(* Logix 5000 project; controller R5_CSS vendor 1 type 14 code 74 rev 19.11; software revision 19.01 *)
// Condensing System

TASK MainTask (continuous, watchdog 500 ms) : MainProgram
TASK MSG (periodic, rate 500 ms, priority 10, watchdog 1000 ms) : POD1_MSG
TASK PIDE (periodic, rate 10 ms, priority 10, watchdog 500 ms) : PIDE   // Advanced PID operations for most important control loops

MODULES
   Local : vendor 1 type 14 code 74 (Compact 0, 1768Ctrl5Slot 0, rev 19.11)
      SLOT_2 : vendor 1 type 7 code 69 (Compact 2, rev 3.1, Input RPI 20 ms)
           Local:2:I.DATA.10   // P205 OVERHEAD CONDENSER PUMP RUN STATUS
      SLOT_3 : vendor 1 type 7 code 69 (Compact 3, rev 3.1, Input RPI 20 ms)
           Local:3:I.DATA.6   // PRIMARY COALESCER SEPARATOR TEMPERATURE CONTROL RUN STATUS
      MVI69 : 1769-MODULE (Compact 1, rev 1.1, Output RPI 2 ms)
      SLOT_11 : 1769-IF8 (Compact 11, rev 1.1, Output RPI 80 ms)
           Local:11:I.CH0DATA   // QUENCH BASIN FLOW TRANSMITTER
           Local:11:I.CH1DATA   // QUENCH FEED FLOW TRANSMITTER
           Local:11:I.CH2DATA   // QUENCH CONDITIONING QUENCH WATER PHASE FLOW TRANSMITTER
           Local:11:I.CH3DATA   // QUENCH TOWER UPPER SPRAY FIT
           Local:11:I.CH4DATA   // QUENCH TOWER LOWER SPRAY FLOW TRANSMITTER
           Local:11:I.CH5DATA   // QUENCH TOWER BASIN LEVEL TRANSMITTER
           Local:11:I.CH6DATA   // QUENCH COALESCING SEPARATOR SECONDARY CHAMBER LEVEL TRANSMITTER
      SLOT_10 : 1769-IF8 (Compact 10, rev 1.1, Output RPI 80 ms)
           Local:10:I.CH3DATA   // QUENCH WATER CONDUCTIVITY TRANSMITTER
           Local:10:I.CH0DATA   // QUENCH BASIN TRANSFER BASIN B TEMPERATURE TRANSMITTER
           Local:10:I.CH1DATA   // COALESCER OIL CHAMBER SHELL TEMPERATURE TRANSMITTER
      SLOT_7 : 1769-IF8 (Compact 7, rev 1.1, Output RPI 80 ms)
           Local:7:I.CH0DATA   // QUENCH TOWER EXIT GAS TEMPERATURE TRANSMITTER
           Local:7:I.CH1DATA   // GTL FROM PRUA TEMPERATURE TRANSMITTER
           Local:7:I.CH2DATA   // GTL FROM PRUB TEMPERATURE TRANSMITTER
           Local:7:I.CH3DATA   // GTL FROM PRUC TEMPERATURE TRANSMITTER
           Local:7:I.CH4DATA   // GTL FROM PRUD TEMPERATURE TRANSMITTER
           Local:7:I.CH5DATA   // HEAT JACKET VENT FROM PRUA TEMPERATURE TRANSMITTER
           Local:7:I.CH6DATA   // HEAT JACKET VENT FROM PRUB TEMPERATURE TRANSMITTER
           Local:7:I.CH7DATA   // HEAT JACKET VENT FROM PRUC TEMPERATURE TRANSMITTER
      SLOT_8 : 1769-IF8 (Compact 8, rev 1.1, Output RPI 80 ms)
           Local:8:I.CH4DATA   // PRIMARY COALESCER SEPARATOR TEMPERATURE TRANSMITTER
           Local:8:I.CH0DATA   // HEAT JACKET VENT FROM PRUD TEMPERATURE TRANSMITTER
           Local:8:I.CH1DATA   // PROCESS WATER POST HX TEMPERATURE TRANSMITTER
           Local:8:I.CH2DATA   // HX COOLING WATER SUPPLY TEMPERATURE TRANSMITTER
           Local:8:I.CH3DATA   // HX COOLING WATER RETURN TEMPERATURE TRANSMITTER
           Local:8:I.CH5DATA   // PRIMARY COALESCER SHELL TEMPERATURE TRANSMITTER
           Local:8:I.CH6DATA   // QUENCH BASIN LIQUID TEMPERATURE TRANSMITTER
           Local:8:I.CH7DATA   // QUENCH BASIN SHELL TEMPERATURE TRANSMITTER
      SLOT_13 : vendor 1 type 10 code 40 (Compact 13, rev 2.1, Output RPI 80 ms)
      SLOT_12 : vendor 1 type 10 code 40 (Compact 12, rev 2.1, Output RPI 80 ms)
      SLOT_4 : 1769-IF8 (Compact 4, rev 1.1, Output RPI 80 ms)
           Local:4:I.CH0DATA   // COALESCER PROCESS IMPURITY FLOW RAW IMPUT
           Local:4:I.CH1DATA   // COALESCER MAKE UP WATER RAW IMPUT
           Local:4:I.CH2DATA   // LOWER QUENCH TOWER PRESSURE TRANSMITTER RAW INPUT
           Local:4:I.CH3DATA   // UPPER QUENCH TOWER PRESSURE TRANSMITTER RAW INPUT
           Local:4:I.CH4DATA   // QUENCH BASIN TRANSFER PUMP SUCTION PRESSURE INDICATOR RAW INPUT
           Local:4:I.CH5DATA   // QUENCH BASIN TRANSFER PUMP DISCHARGE PRESSURE RAW INPUT
           Local:4:I.CH6DATA   // PRE HX LOW PRESSURE TRANSMITTER RAW INPUT
           Local:4:I.CH7DATA   // POST HX LOW PRESSURE TRANSMITTER RAW INPUT
      SLOT_9 : 1769-IF8 (Compact 9, rev 1.1, Output RPI 80 ms)
           Local:9:I.CH0DATA   // OVERHEAD CONDENSER CHILLED WATER TEMPERATURE TRANSMITTER
           Local:9:I.CH1DATA   // OVERHEAD CONDENSER BASIN TEMPERATURE TRANSMITTER
           Local:9:I.CH2DATA   // OVERHEAD CONDENSER CHILLED WATER SUPPLY TEMPERATURE
           Local:9:I.CH3DATA   // OVERHEAD CONDENSED CHILLED WATER RETURN TEMPERATURE TRANSMITTER
           Local:9:I.CH4DATA   // COALESCER OIL CHAMBER SHELL TEMPERATURE TRANSMITTER
           Local:9:I.CH5DATA   // COALESCER OIL CHAMBER TRANSFER PUMP A TEMPERATURE TRANSMITTER
           Local:9:I.CH6DATA   // COALESCER OIL CHAMBER TRANSFER PUMP B TEMPERATURE TRANSMITTER
           Local:9:I.CH7DATA   // QUENCH BASIN TRANSFER BASIN A TEMPERATURE TRANSMITTER
      SLOT_5 : 1769-IF8 (Compact 5, rev 1.1, Output RPI 80 ms)
           Local:5:I.CH4DATA   // VACUUM SYSTEM PRESSURE TRANSMITTER RAW INPUT
           Local:5:I.CH5DATA   // HX COOLING WATER FLOW TRANMITTER
           Local:5:I.CH6DATA   // OVERHEAD CONDENSER CHILLED WATER FLOW TRANSMITTER RAW INPUT
           Local:5:I.CH7DATA   // VENT HEADER PRESSURE TRANSMITTER RAW INPUT
      SLOT_14 : vendor 1 type 7 code 73 (Compact 14, rev 3.1, Output RPI 20 ms)
           Local:14:O.DATA.4   // HS302B P302B Oil Transfer Pump Start Relay
           Local:14:O.DATA.5   // HS205 P205 Overhead Condenser Basin Transfer Start
           Local:14:O.DATA.25   // MP-113 Start
           Local:14:O.DATA.26   // Alarm Horn (Future)
           Local:14:O.DATA.12   // FCV141 PLANT RAW WATER INLET TO QUENCH TOWER ENERGIZE TO OPEN
           Local:14:O.DATA.0   // Loss of Panel Purge Indicator Light
           Local:14:O.DATA.1   // Spare
           Local:14:O.DATA.2   // Spare
           Local:14:O.DATA.14   // HS104B Valve P101B Quench Transfer FAIL OPEN ENERGISE TO CLOSE
           Local:14:O.DATA.16   // HS313 Primary Settler Heat Controller
           Local:14:O.DATA.3   // HS302A P302A Oil Transfer Pump Start Relay
           Local:14:O.DATA.7   // HS_MP112 Quench Transfer Metal Treat Meter Pump #2 Start
           Local:14:O.DATA.6   // HS_MP113 Quench Transfer Metal Treat Meter Pump #1 Start
           Local:14:O.DATA.17   // JC306 or HS306A OIL CHAMBER SETTLER HEAT OUTPUT START
           Local:14:O.DATA.9   // HS_MP411 Quench Condition Metal Treat Meter Pump #2 Start (future)
           Local:14:O.DATA.8   // HS_MP410 Quench Condition Metal Treat Meter Pump #1 Start (future)
           Local:14:O.DATA.10   // HS315A VALVE P303A DISCHARGE FAIL OPEN ENERGIZE TO CLOSE
           Local:14:O.DATA.11   // HS315B VALVE P303B DISCHARGE FAIL OPEN ENERGIZE TO CLOSE
           Local:14:O.DATA.13   // HS104A Valve P101A Quench Transfer FAIL OPEN ENERGISE TO CLOSE
           Local:14:O.DATA.15   // Spare
           Local:14:O.DATA.18   // HS114B Quench Tower Heat Controller Hand Switch
           Local:14:O.DATA.20   // HS433B Valve HX B COOLING WATER ENERGIZE TO CLOSE
           Local:14:O.DATA.22   // HS431B Inlet Valve HX B PROCESS ENERGIZE TO CLOSE
           Local:14:O.DATA.21   // HS431A Inlet Valve HX A PROCESS ENERGIZE TO CLOSE
           Local:14:O.DATA.19   // HS433A Valve HX A COOLING WATER ENERGIZE TO CLOSE
           Local:14:O.DATA.23   // FCV410 Quench Basin Level Transmitter Hot Water Flush
           Local:14:O.DATA.24   // MV361 Sec/Ter Coalsce Chamber CrossOver Valve H3 Occupancy
           Local:14:O.DATA.27   // MV115B Basin Water Heater Valve
      SLOT_6 : 1769-IF8 (Compact 6, rev 1.1, Output RPI 80 ms)
           Local:6:I.CH0DATA   // OVERHEAD CONDENSER BASIN LEVEL TRANSMITTER RAW INPUT
           Local:6:I.CH1DATA   // COALESCER OIL CHAMBER LEVEL TRANSMITTER RAW INPUT
           Local:6:I.CH3DATA   // OVERHEAD CONDENSER CHILLED WATER TEMPERATURE TRANSMITTER RAW INPUT
      CSS_ENET : 1768-ENBT (1768 1, Ethernet 192.168.20.70, rev 4.1)
         P303B : ETHERNET-MODULE (Ethernet 192.168.20.75, rev 1.1, Output RPI 10 ms)
              P303B:I.DATA[2]   // Status Bits (Continued)
              P303B:I.DATA[2].9   // Local/Remote Keypad Status 0=Local 1-=Remote
              P303B:I.DATA[1]   // Current RPM
              P303B:I.DATA[0].0   // Faulted
              P303B:I.DATA[0].1   // Warning
              P303B:I.DATA[0].2   // Running in Forward
              P303B:I.DATA[0].3   // Running in Reverse
              P303B:I.DATA[0].4   // Ready
              P303B:I.DATA[0].5   // Ctrl from Net
              P303B:I.DATA[0].6   // Ref from Net
              P303B:I.DATA[0].7   // At Reference
              P303B:I.DATA[0]   // Status Bits
              P303B:I.DATA   // Instance 171
              P303B:I.DATA[4]   // Current Amps
              P303B:O.DATA   // Instance 21
              P303B:O.DATA[0]   // Command Bits
              P303B:O.DATA[0].0   // Run Forward Command
              P303B:O.DATA[0].1   // Run Reverse Command
              P303B:O.DATA[0].2   // Fault Reset
              P303B:O.DATA[1]   // RPM Speed Refernce
         P303A : ETHERNET-MODULE (Ethernet 192.168.20.74, rev 1.1, Output RPI 10 ms)
              P303A:I.DATA[0]   // Status Bits
              P303A:I.DATA   // Instance 171
              P303A:I.DATA[1]   // Current RPM
              P303A:I.DATA[2]   // Status Bits (Continued)
              P303A:I.DATA[4]   // Current Amps
              P303A:I.DATA[0].0   // Faulted
              P303A:I.DATA[0].1   // Warning
              P303A:I.DATA[0].2   // Running in Forward
              P303A:I.DATA[0].3   // Running in Reverse
              P303A:I.DATA[0].4   // Ready
              P303A:I.DATA[0].5   // Ctrl from Net
              P303A:I.DATA[0].6   // Ref from Net
              P303A:I.DATA[0].7   // At Reference
              P303A:I.DATA[2].9   // Local/Remote Keypad Status 0=Local 1-=Remote
              P303A:O.DATA   // Instance 21
              P303A:O.DATA[0]   // Command Bits
              P303A:O.DATA[0].1   // Run Reverse Command
              P303A:O.DATA[0].2   // Fault Reset
              P303A:O.DATA[1]   // RPM Speed Reference
              P303A:O.DATA[0].0   // Run Forward Command
         P101A : ETHERNET-MODULE (Ethernet 192.168.20.72, rev 1.1, Output RPI 10 ms)
              P101A:I.DATA[2]   // Status Bits (Continued)
              P101A:I.DATA[4]   // Current Amps
              P101A:I.DATA[0].5   // Ctrl from Net
              P101A:I.DATA[0].3   // Running In Reverse
              P101A:I.DATA[0].2   // Running In Forward
              P101A:I.DATA[0]   // Status Bits
              P101A:I.DATA   // Instance 171
              P101A:I.DATA[0].0   // Faulted
              P101A:I.DATA[0].1   // Warning
              P101A:I.DATA[0].4   // Ready
              P101A:I.DATA[0].6   // Ref from Net
              P101A:I.DATA[0].7   // At Refernce
              P101A:I.DATA[1]   // Current RPM
              P101A:I.DATA[2].9   // Local/Remote Keypad Status 0=Local 1=Remote
              P101A:O.DATA[0].8   // na
              P101A:O.DATA[1]   // RPM Speed Reference
              P101A:O.DATA[0].0   // Run Forward Command
              P101A:O.DATA[0].1   // Run Reverse Command
              P101A:O.DATA[0].2   // Fault Reset
              P101A:O.DATA[0].5   // NetCtrl
              P101A:O.DATA[0]   // Command Bits
              P101A:O.DATA[0].6   // NetRef
              P101A:O.DATA[0].10   // na
              P101A:O.DATA[0].9   // na
              P101A:O.DATA[0].11   // na
              P101A:O.DATA[0].12   // na
              P101A:O.DATA[0].13   // na
              P101A:O.DATA[0].14   // na
              P101A:O.DATA[0].15   // na
              P101A:O.DATA[0].7   // na
              P101A:O.DATA[0].4   // na
              P101A:O.DATA[0].3   // na
              P101A:O.DATA   // Instance 21
         P101B : ETHERNET-MODULE (Ethernet 192.168.20.73, rev 1.1, Output RPI 10 ms)
              P101B:I.DATA   // Instance 171
              P101B:I.DATA[0]   // Status Bits
              P101B:I.DATA[0].0   // Faulted
              P101B:I.DATA[0].1   // Warning
              P101B:I.DATA[0].2   // Running in Forward
              P101B:I.DATA[0].3   // Running in Reverse
              P101B:I.DATA[0].4   // Ready
              P101B:I.DATA[0].5   // Ctrl from Net
              P101B:I.DATA[0].6   // Ref from Net
              P101B:I.DATA[0].7   // At Reference
              P101B:I.DATA[1]   // Current RPM
              P101B:I.DATA[2]   // Status Bits (Continued)
              P101B:I.DATA[4]   // Current Amps
              P101B:I.DATA[2].9   // Local/Remote Keypad Status 0=Local 1=Remote
              P101B:O.DATA[1]   // RPM Speed Reference
              P101B:O.DATA[0]   // Command Bits
              P101B:O.DATA[0].0   // Run Forward Command
              P101B:O.DATA[0].1   // Run Reverse Command
              P101B:O.DATA[0].2   // Fault Reset
              P101B:O.DATA   // Instance 21
END_MODULES

TYPE AnalogControl :
STRUCT
   AUTO : BOOL;
   MANUAL : BOOL;
   MAN_SP : REAL;
   AUTO_SP : REAL;
   CO : REAL;
   FB : REAL;
   PID_CO : REAL;
   PV_SETPOINT : REAL;
   PV : REAL;
   HC_FAULT : BOOL;
   RUN_STATUS : BOOL;   // Boolean feedback of the running status of the associated output
   START : BOOL;   // Master logical bit used to enable an associated output
   XA_Low : BOOL;   // Signal failure (Low counts)
   XA_High : BOOL;   // Signal failure (High counts)
   RawCounts : DINT;   // Raw integer from input card
   FailMode : DINT;   // 0=raw, 1=hold last, 2=safe state
   SafeState : REAL;   // Used to hold an analog value in the event of a failed instrument
   AI_Anal : AI_Analysis;   // Used to manage an analog input to determine scaled value and loss of signal alarms
   InputMin : DINT;   // Input card lower counts i.e. 4mA - 4000 counts
   InputMax : DINT;   // Input card upper counts i.e. 20mA - 20000 counts
   ScaledMin : REAL;   // Analog low Engineering unit i.e. 4mA - 0 psi
   ScaledMax : REAL;   // Analog High Engineering unit i.e. 20mA - 100 psi
   OutputMin : DINT;   // Output card lower counts i.e. 4mA - 4000 counts
   OutputMax : DINT;   // Output card upper counts i.e. 4mA - 4000 counts
   AlarmsSetDetaults : BOOL;   // reloads the default alarm limits and setup
   Simulate : BOOL;   // 0=raw counts from Input card, 1=simulation raw counts
   RawCountsSim : DINT;   // raw count simulation from HMI/Programmer
   DifferenceExists : BOOL;
   LoadDefaults : BOOL;
   StoreDefaults : BOOL;
END_STRUCT
END_TYPE

TYPE ANALYTICAL :
STRUCT
   AUTO : BOOL;
   MANUAL : BOOL;
   MAN_SP : REAL;
   AUTO_SP : REAL;
   CO : REAL;
   FB : REAL;
   PID_CO : REAL;
   PV_SETPOINT : REAL;
   AT : REAL;
   AALL_SP : REAL;
   AAL_SP : REAL;
   AAH_SP : REAL;
   AAHH_SP : REAL;
   ALL_DEV : REAL;
   AL_DEV : REAL;
   AH_DEV : REAL;
   AHH_DEV : REAL;
   AALL : BOOL;
   AAL : BOOL;
   AAH : BOOL;
   AAHH : BOOL;
   ALL_TMR : TIMER;
   AL_TMR : TIMER;
   AH_TMR : TIMER;
   AHH_TMR : TIMER;
   XA : BOOL;   // LOSS OF SIGNAL
   Forced : BOOL;   // Override actual signal with forced value
   ForcedValue : REAL;   // used with the Forced bit
   XA_Low : BOOL;   // Signal failure (Low counts)
   XA_High : BOOL;   // Signal failure (High counts)
   RawCounts : DINT;   // Raw integer from input card
   FailMode : DINT;   // 0=raw, 1=hold last, 2=safe state
   SafeState : REAL;   // Used to hold an analog value in the event of a failed instrument
   AI_Anal : AI_Analysis;   // Used to manage an analog input to determine scaled value and loss of signal alarms
   InputMin : DINT;   // Input card lower counts i.e. 4mA - 4000 counts
   InputMax : DINT;   // Input card upper counts i.e. 20mA - 20000 counts
   ScaledMin : REAL;   // Analog low Engineering unit i.e. 4mA - 0 psi
   ScaledMax : REAL;   // Analog High Engineering unit i.e. 20mA - 100 psi
   OutputMin : DINT;   // Output card lower counts i.e. 4mA - 4000 counts
   OutputMax : DINT;   // Output card upper counts i.e. 4mA - 4000 counts
   AlarmsSetDetaults : BOOL;   // reloads the default alarm limits and setup
   Simulate : BOOL;   // 0=raw counts from Input card, 1=simulation raw counts
   RawCountsSim : DINT;   // raw count simulation from HMI/Programmer
   DifferenceExists : BOOL;   // 0 - current settings are equal to default 1 = current settings differ from default
   LoadDefaults : BOOL;   // set to 1 to load from default settings
   StoreDefaults : BOOL;   // set to 1 to save current settings into default placeholder
   PV : REAL;   // Real signal from instrument in engineering units
END_STRUCT
END_TYPE

TYPE FAULTRECORD :
STRUCT
   TIMELOW : DINT;
   TIMEHIGH : DINT;
   TYPE : INT;
   CODE : INT;
   INFO : DINT[8];
END_STRUCT
END_TYPE

TYPE FLOW_CONTROL :
STRUCT
   AUTO : BOOL;
   MANUAL : BOOL;
   MAN_SP : REAL;
   AUTO_SP : REAL;
   CO : REAL;
   FB : REAL;
   PID_CO : REAL;
   PV_SETPOINT : REAL;
   FT : REAL;
   FALL_SP : REAL;
   FAL_SP : REAL;
   FAH_SP : REAL;
   FAHH_SP : REAL;
   FALL_DEV : REAL;
   FAL_DEV : REAL;
   FAH_DEV : REAL;
   FAHH_DEV : REAL;
   FALL : BOOL;
   FAL : BOOL;
   FAH : BOOL;
   FAHH : BOOL;
   FALL_TMR : TIMER;
   FAL_TMR : TIMER;
   FAH_TMR : TIMER;
   FAHH_TMR : TIMER;
   XA : BOOL;   // OUT OF RANGE (LOW)
   Forced : BOOL;   // Override actual signal with forced value
   ForcedValue : REAL;   // used with the Forced bit
   XA_Low : BOOL;   // Signal failure (Low counts)
   XA_High : BOOL;   // Signal failure (High counts)
   RawCounts : DINT;   // Raw integer from input card
   FailMode : DINT;   // 0=raw, 1=hold last, 2=safe state
   SafeState : REAL;   // Used to hold an analog value in the event of a failed instrument
   AI_Anal : AI_Analysis;   // Used to manage an analog input to determine scaled value and loss of signal alarms
   InputMin : DINT;   // Input card lower counts i.e. 4mA - 4000 counts
   InputMax : DINT;   // Input card upper counts i.e. 20mA - 20000 counts
   ScaledMin : REAL;   // Analog low Engineering unit i.e. 4mA - 0 psi
   ScaledMax : REAL;   // Analog High Engineering unit i.e. 20mA - 100 psi
   OutputMin : DINT;   // Output card lower counts i.e. 4mA - 4000 counts
   OutputMax : DINT;   // Output card upper counts i.e. 4mA - 4000 counts
   AlarmsSetDetaults : BOOL;   // reloads the default alarm limits and setup
   Simulate : BOOL;   // 0=raw counts from Input card, 1=simulation raw counts
   RawCountsSim : DINT;   // raw count simulation from HMI/Programmer
   DifferenceExists : BOOL;   // 0 - current settings are equal to default 1 = current settings differ from default
   LoadDefaults : BOOL;   // set to 1 to load from default settings
   StoreDefaults : BOOL;   // set to 1 to save current settings into default placeholder
   PV : REAL;   // Real signal from instrument in engineering units
END_STRUCT
END_TYPE

TYPE HARTAutoPoll :
STRUCT
   Auto_Poll_CMD_Status : SINT;
   Last_Status_Byte : SINT;
   Last_Second_Status_Byte : SINT;
   Manufacture_ID_Code : SINT;
   Device_Type_Code : SINT;
   Min_Preambles : SINT;
   Universal_CMD_Major : SINT;
   Device_Rev_Level : SINT;
   Software_Rev_Level : SINT;
   Hardware_Rev_Level : SINT;
   Device_Flags : SINT;
   Device_ID : SINT[3];
   Min_Preambles_Resp : SINT;
   Max_Number_Devices : SINT;
   Config_Change_Count : INT;
   Ext_Dev_Status : SINT;
   Primary_Var_Units : SINT;
   Secondary_Var_Units : SINT;
   Tertiary_Var_Units : SINT;
   Quaternary_Var_Units : SINT;
   Tag_Name : SINT[8];
   Descriptor : SINT[16];
   Tag_Descriptor_Data : SINT[3];
   Transd_Serial_Num : SINT[3];
   Transd_limits : SINT;
   PV_Alarms : SINT;
   PV_Transfer : SINT;
   PV_URLLRV_Units : SINT;
   Write_Protection_Code : SINT;
   Private_Label_Code : SINT;
   PV_Analog_Ch_Flag : SINT;
   PV_value : REAL;
   SV_value : REAL;
   TV_value : REAL;
   QV_value : REAL;
   U_trans_limit : REAL;
   L_trans_limit : REAL;
   Min_span : REAL;
   PV_URV : REAL;
   PV_LRV : REAL;
   PV_damp : REAL;
END_STRUCT
END_TYPE

TYPE HARTBackplane :
STRUCT
   LastRead : INT;
   LastWrite : INT;
   BlockIndex : INT;
END_STRUCT
END_TYPE

TYPE HARTCHStat :
STRUCT
   State : INT;
   Comm_State : INT;
   Dev_stat : INT;
   Dev_in_poll : INT;
   Dev_long : INT;
   Cur_cmd : INT;
   Cmd_req : INT;
   Cmd_resp : INT;
   Cfg_Err : INT;
   CurErr : INT;
   LastErr : INT;
END_STRUCT
END_TYPE

TYPE HARTData :
STRUCT
   HART_IN_Float_vals : REAL[100];
   HART_IN_Int_vals : INT[500];
   HART_OUT_Float_vals : REAL[100];
   HART_OUT_Int_vals : INT[500];
END_STRUCT
END_TYPE

TYPE HARTModuleDef :
STRUCT
   GenStat : HARTStat;
   BP : HARTBackplane;
   Auto_Poll : HARTAutoPoll[10];
   ByteData : SINT[1000];
   BlockTransferSize : INT;
END_STRUCT
END_TYPE

TYPE HARTStat :
STRUCT
   Scan_Cnt : INT;
   Product_Name : SINT[4];
   Rev_Level : SINT[4];
   Op_Sys : SINT[4];
   Run_Number : SINT[4];
   Blk_Rd_Count : INT;
   Blk_Wr_Count : INT;
   Blk_Parse_Cnt : INT;
   Blk_Resv : INT;
   Blk_Cmd : INT;
   Blk_Err : INT;
   ChStat : HARTCHStat[2];
END_STRUCT
END_TYPE

TYPE IP :
STRUCT
   IP1 : SINT;
   IP2 : SINT;
   IP3 : SINT;
   IP4 : SINT;
   SN1 : SINT;
   SN2 : SINT;
   SN3 : SINT;
   SN4 : SINT;
   GW1 : SINT;
   GW2 : SINT;
   GW3 : SINT;
   GW4 : SINT;
   PNS1 : SINT;
   PNS2 : SINT;
   PNS3 : SINT;
   PNS4 : SINT;
   SNS1 : SINT;
   SNS2 : SINT;
   SNS3 : SINT;
   SNS4 : SINT;
   EMPTY : INT;
   DN : SINT[48];
END_STRUCT
END_TYPE

TYPE LEVEL_CONTROL :
STRUCT
   AUTO : BOOL;
   MANUAL : BOOL;
   MAN_SP : REAL;
   AUTO_SP : REAL;   // PUMP START SET POINT
   CO : REAL;
   FB : REAL;
   PID_CO : REAL;
   PV_SETPOINT : REAL;
   LT : REAL;
   LALL_SP : REAL;
   LAL_SP : REAL;
   LAH_SP : REAL;
   LAHH_SP : REAL;
   LDAH_SP : REAL;   // LDAH SETPOING
   LALL_DEV : REAL;
   LAL_DEV : REAL;
   LAH_DEV : REAL;
   LAHH_DEV : REAL;
   LDAH_DEV : REAL;   // LDAH DEVIATION
   LDAH_DIFF : REAL;   // LDAH DIFFERENCE
   LALL : BOOL;
   LAL : BOOL;
   LAH : BOOL;
   LAHH : BOOL;
   LDAH : BOOL;   // HIGH DIFFERENTIAL
   LALL_TMR : TIMER;
   LAL_TMR : TIMER;
   LAH_TMR : TIMER;
   LAHH_TMR : TIMER;
   LDAH_TMR : TIMER;   // HIGH DIFFERENTIAL TIMVER
   XA : BOOL;   // OUT OF RANGE SIGNAL
   Forced : BOOL;   // Override actual signal with forced value
   ForcedValue : REAL;   // used with the Forced bit
   XA_Low : BOOL;   // Signal failure (Low counts)
   XA_High : BOOL;   // Signal failure (High counts)
   RawCounts : DINT;   // Raw integer from input card
   FailMode : DINT;   // 0=raw, 1=hold last, 2=safe state
   SafeState : REAL;   // Used to hold an analog value in the event of a failed instrument
   AI_Anal : AI_Analysis;   // Used to manage an analog input to determine scaled value and loss of signal alarms
   InputMin : DINT;   // Input card lower counts i.e. 4mA - 4000 counts
   InputMax : DINT;   // Input card upper counts i.e. 20mA - 20000 counts
   ScaledMin : REAL;   // Analog low Engineering unit i.e. 4mA - 0 psi
   ScaledMax : REAL;   // Analog High Engineering unit i.e. 20mA - 100 psi
   OutputMin : DINT;   // Output card lower counts i.e. 4mA - 4000 counts
   OutputMax : DINT;   // Output card upper counts i.e. 4mA - 4000 counts
   AlarmsSetDetaults : BOOL;   // reloads the default alarm limits and setup
   Simulate : BOOL;   // 0=raw counts from Input card, 1=simulation raw counts
   RawCountsSim : DINT;   // raw count simulation from HMI/Programmer
   DifferenceExists : BOOL;   // 0 - current settings are equal to default 1 = current settings differ from default
   LoadDefaults : BOOL;   // set to 1 to load from default settings
   StoreDefaults : BOOL;   // set to 1 to save current settings into default placeholder
   PV : REAL;   // Real signal from instrument in engineering units
END_STRUCT
END_TYPE

TYPE MAJOR_FAULT :
STRUCT
   TYPE : INT;
   CODE : INT;
   INFO : DINT[8];   // [0] = Task [1] = Program [2] = Routine [3] = Address [4]-[7] not used
END_STRUCT
END_TYPE

TYPE MSG_CommsPath :
STRUCT
   Prefix : STRING;   // This is the standard hex prefix to be used to build the path
   NodeNum : DINT;   // This is the configurable node number
   NodeStr : STRING;   // this is the node number represented as a string
   Path : STRING;   // this is the complete path
END_STRUCT
END_TYPE

TYPE PRESSURE_CONTROL :
STRUCT
   AUTO : BOOL;
   MANUAL : BOOL;
   MAN_SP : REAL;
   AUTO_SP : REAL;
   CO : REAL;
   FB : REAL;
   PID_CO : REAL;
   PV_SETPOINT : REAL;
   PT : REAL;
   PDAHH_DIFF : REAL;   // PDAHH DIFFERENCE
   PDAH_DIFF : REAL;   // PDAH DIFFERENCE
   PALL_SP : REAL;
   PAL_SP : REAL;
   PAH_SP : REAL;
   PAHH_SP : REAL;
   PDAH_SP : REAL;   // HIGH DIFFERENTIAL SETPOINT
   PDAHH_SP : REAL;   // PDAHH DIFF SP
   PALL_DEV : REAL;
   PAL_DEV : REAL;
   PAH_DEV : REAL;
   PAHH_DEV : REAL;
   PDAH_DEV : REAL;   // HIGH DIFFERENTIAL ALARM CLEAR
   PDAHH_DEV : REAL;   // HI HI DIFFERENTIAL ALARM CLEAR
   PALL : BOOL;
   PAL : BOOL;
   PAH : BOOL;
   PAHH : BOOL;
   PDAH : BOOL;   // HIGH DIFFERENTIAL ALARM
   PDAHH : BOOL;   // DIFFERENTIAL ALARM HI HI
   PALL_TMR : TIMER;
   PAL_TMR : TIMER;
   PAH_TMR : TIMER;
   PDAH_TMR : TIMER;   // HIGH DIFFERENTIAL DEBOUNCE TIMER
   PAHH_TMR : TIMER;
   PDAHH_TMR : TIMER;   // HI HI DIFFERENTIAL DEBOUNCE TIMER
   XA : BOOL;   // LOSS OF SIGNAL
   XA_Low : BOOL;   // Signal failure (Low counts)
   XA_High : BOOL;   // Signal failure (High counts)
   RawCounts : DINT;   // Raw integer from input card
   FailMode : DINT;   // 0=raw, 1=hold last, 2=safe state
   SafeState : REAL;   // Used to hold an analog value in the event of a failed instrument
   AI_Anal : AI_Analysis;   // Used to manage an analog input to determine scaled value and loss of signal alarms
   InputMin : DINT;   // Input card lower counts i.e. 4mA - 4000 counts
   InputMax : DINT;   // Input card upper counts i.e. 20mA - 20000 counts
   ScaledMin : REAL;   // Analog low Engineering unit i.e. 4mA - 0 psi
   ScaledMax : REAL;   // Analog High Engineering unit i.e. 20mA - 100 psi
   OutputMin : DINT;   // Output card lower counts i.e. 4mA - 4000 counts
   OutputMax : DINT;   // Output card upper counts i.e. 4mA - 4000 counts
   AlarmsSetDetaults : BOOL;   // reloads the default alarm limits and setup
   Simulate : BOOL;   // 0=raw counts from Input card, 1=simulation raw counts
   RawCountsSim : DINT;   // raw count simulation from HMI/Programmer
   DifferenceExists : BOOL;   // 0 - current settings are equal to default 1 = current settings differ from default
   LoadDefaults : BOOL;   // set to 1 to load from default settings
   StoreDefaults : BOOL;   // set to 1 to save current settings into default placeholder
   PV : REAL;   // Real signal from instrument in engineering units
END_STRUCT
END_TYPE

TYPE PUMP_CONTROL :
STRUCT
   QAS_IAS : BOOL;
   QI_AUTO : BOOL;
   QI_MANUAL : BOOL;
   QI_LEAD : BOOL;   // LEAD STATUS
   QI_TRANSFER_LEAD : BOOL;   // HMI REQUEST LEAD
   QI_RUN_STATUS : BOOL;
   START : BOOL;
   LAL_ENABLE : BOOL;
   TAL_ENABLE : BOOL;
   LOCAL_STATUS : BOOL;   // LOCAL/AUTO STATUS AT VFD Keypad 0=Local 1=Auto
   YI_LEAD : BOOL;   // LEAD CHANGE ALERT TO SUP STATION
   XA : BOOL;   // LOSS OF SIGNAL
   ACK : BOOL;   // PUMP FAULT ACKNOWLEDGE
   DISABLE : BOOL;   // PUMP DISABLE
   QI_DAYS : INT;   // PUMP RUN DAYS TOTALIZER
   QI_HOURS : INT;   // PUMP RUN HOURS TOTALIZER
   CO : INT;   // CONTROL OUTPUT TO THE PUMP
   LEAD_DAYS_SP : INT;
   SIC : INT;
   FB : INT;   // FEEDBACK RPM
   IAS_SP : REAL;   // Low Current Alarm Setpoint
   SIC_MAN_SP : REAL;
   SIC_AUTO_SP : REAL;
   RAMP_SP : REAL;
   CO_HZ : REAL;   // HERTZ OUTPUT
   FB_HZ : REAL;   // FEEBACK
   EI : REAL;   // Current Amps
   TAL_SP : REAL;
   CUMULATIVE_TM : REAL;
   QAS_IAS_TMR : TIMER;   // Pump Fault Timer
   TAL_TMR : TIMER;
   LEAD_XFER_TMR : TIMER;
   RUN_HRS : TIMER;
   SPEED_DELAY : TIMER;
   START_DELAY : TIMER;   // DELAY TO START PUMP )TO OPEN VALVE ETC.
   ENET : BOOL;   // VFD ENET STATUS
   ENET_STAT : DINT;   // EMAIL STATUS SB BETWEEN 16384 and 20479 ( h4000 -h4999)
   ENET_FAULT : DINT;   // ENET FAULT
   ENET_REG_FAULT : DINT;   // ENET REGISTERED FAULT
   ENET_DATE_TIME : DINT[9];   // FAULT DATE TIME
   Power : REAL;   // Current Power in kwatts
   Energy : REAL;   // Total Energy in kW-hr
   kWh_Tmr : TIMER;   // Energy Totalizer sample timer
   kWh_ResetPB : BOOL;   // HMI Reset Energy totals
   kWh_SampleTime : REAL;   // in seconds
   kWh_TimeMultiplier : REAL;   // derived from the SampleTime to ensure kW-Hr units
END_STRUCT
END_TYPE

TYPE TCPGetAllConfig :
STRUCT
   IPAddress : DINT;
   SubNetMask : DINT;
   Gateway : DINT;
   NameServer1 : DINT;
   NameServer2 : DINT;
   DomainName : STRING;
END_STRUCT
END_TYPE

TYPE TCPSetAllConfig :
STRUCT
   IPAddress : DINT;   // I/P Address
   SubNetMask : DINT;   // SubNet Mask
   Gateway : DINT;   // Gateway I/P address
   NameServer1 : DINT;   // Primary DNS Server Address
   NameServer2 : DINT;   // Secondary DNS Server Address
   DomainName : SINT[50];
END_STRUCT
END_TYPE

TYPE TEMP_CONTROL :
STRUCT
   AUTO : BOOL;
   MANUAL : BOOL;
   MAN_SP : REAL;
   AUTO_SP : REAL;
   CO : REAL;
   FB : REAL;
   PID_CO : REAL;
   PV_SETPOINT : REAL;
   TT : REAL;
   TALL_SP : REAL;
   TAL_SP : REAL;
   TAH_SP : REAL;
   TAHH_SP : REAL;
   TDAH_SP : REAL;   // DIFFERENTIAL ALARM SETPOINT
   DIFFERENCE : REAL;   // DIFFERTIAL RESULT
   TALL : BOOL;
   TAL : BOOL;
   TAH : BOOL;
   TAHH : BOOL;
   TDAH : BOOL;   // DIFFERENTIAL ALARM
   TALL_TMR : TIMER;
   TAL_TMR : TIMER;
   TAH_TMR : TIMER;
   TAHH_TMR : TIMER;
   TDAH_TMR : TIMER;   // DIFFERENTIAL ALARM DEBOUNCE TIMER
   TAHH_DEV : REAL;
   TAH_DEV : REAL;
   TAL_DEV : REAL;
   TALL_DEV : REAL;
   TDAH_DEV : REAL;   // ALARM CLEAR SP
   HC_FAULT : BOOL;
   RUN_STATUS : BOOL;
   START : BOOL;   // START COMMAND
   XA : BOOL;   // LOSS OF SIGNAL TRANSMITTER
   Forced : BOOL;   // Override actual signal with forced value
   ForcedValue : REAL;   // used with the Forced bit
   XA_Low : BOOL;   // Signal failure (Low counts)
   XA_High : BOOL;   // Signal failure (High counts)
   RawCounts : DINT;   // Raw integer from input card
   FailMode : DINT;   // 0=raw, 1=hold last, 2=safe state
   SafeState : REAL;   // Used to hold an analog value in the event of a failed instrument
   AI_Anal : AI_Analysis;   // Used to manage an analog input to determine scaled value and loss of signal alarms
   InputMin : DINT;   // Input card lower counts i.e. 4mA - 4000 counts
   InputMax : DINT;   // Input card upper counts i.e. 20mA - 20000 counts
   ScaledMin : REAL;   // Analog low Engineering unit i.e. 4mA - 0 psi
   ScaledMax : REAL;   // Analog High Engineering unit i.e. 20mA - 100 psi
   OutputMin : DINT;   // Output card lower counts i.e. 4mA - 4000 counts
   OutputMax : DINT;   // Output card upper counts i.e. 4mA - 4000 counts
   AlarmsSetDetaults : BOOL;   // reloads the default alarm limits and setup
   Simulate : BOOL;   // 0=raw counts from Input card, 1=simulation raw counts
   RawCountsSim : DINT;   // raw count simulation from HMI/Programmer
   DifferenceExists : BOOL;   // 0 - current settings are equal to default 1 = current settings differ from default
   LoadDefaults : BOOL;   // set to 1 to load from default settings
   StoreDefaults : BOOL;   // set to 1 to save current settings into default placeholder
   PV : REAL;   // Real signal from instrument in engineering units
   kWh_Tmr : TIMER;   // Energy Totalizer sample timer
   kWh_ResetPB : BOOL;   // HMI Reset Energy totals
   kWh_SampleTime : REAL;   // in seconds
   kWh_TimeMultiplier : REAL;   // derived from the SampleTime to ensure kW-Hr units
   Power : REAL;   // Current Power in kwatts
   Energy : REAL;   // Total Energy in kW-hr
   HeaterRating_kWh : REAL;   // in kW-hr
END_STRUCT
END_TYPE

TYPE TheTotalizer :
STRUCT
   Enable : BOOL;   // Continue to Totalize
   TotalSecTmr : TIMER;
   Minutes : REAL;   // Current Totalize time in min
   MinutesLast : REAL;   // Last Totalize Time in Min
   ONS : DINT;   // OneShot Bits
   ResetPB : BOOL;   // Reset Push Button from HMI
   Totalizer : Totalize;
   Total : REAL;   // Total (the money shot)
   Disable : BOOL;   // Simulating a flow valve
   Last_Add : REAL;   // Last total adder
   Reset : BOOL;   // Internally used to reset the totalizer
   Seconds : DINT;   // Time in seconds
   Hours : REAL;
   HoursLast : REAL;
END_STRUCT
END_TYPE

TYPE ValveControl_TwoWay :
STRUCT
   Status : BOOL;   // Status of the Valve Output 0=Closed 1=Open
   Manual : BOOL;   // Manual Output Command 1=Energized
   OpenStat : BOOL;   // Postion Switch
   ClosedStat : BOOL;   // Postion Switch
   Auto : BOOL;   // 0=Manual 1=Auto
END_STRUCT
END_TYPE

ADD_ON_INSTRUCTION AI_Analysis   (* revision 1.0 *)
VAR_OUTPUT
   XmtrOut : REAL; {access Read Only, required}
END_VAR
VAR_INPUT
   RawCounts : DINT; {required}
   SafeState : REAL; {required}
END_VAR
VAR_OUTPUT
   SigLossHigh : BOOL; {required}
   SigLossLow : BOOL; {required}
END_VAR
VAR_INPUT
   FailMode : DINT; {required}   // 0=raw, 1=last state, 2=safe state
   SigLossHighSP : DINT; {required}
   SigLossLowSP : DINT; {required}
   InputMin : REAL; {required}
   InputMax : REAL; {required}
   ScaledMin : REAL; {required}
   ScaledMax : REAL; {required}
   Simulate : BOOL; {required}
   RawCountsSim : DINT; {access None, required}
END_VAR
VAR
   SigLoss : BOOL; {access None}
   LastState : REAL; {access None}
   MyXmtrSCP : SCLP; {access None}
   MyRawCounts : DINT; {access None}
   SigLossLowTmr : TIMER := (PRE := 2000); {access None}
   SigLossHighTmr : TIMER := (PRE := 2000); {access None}
   HoldLast : BOOL; {access None}
END_VAR

ROUTINE Logic   (* ladder *)
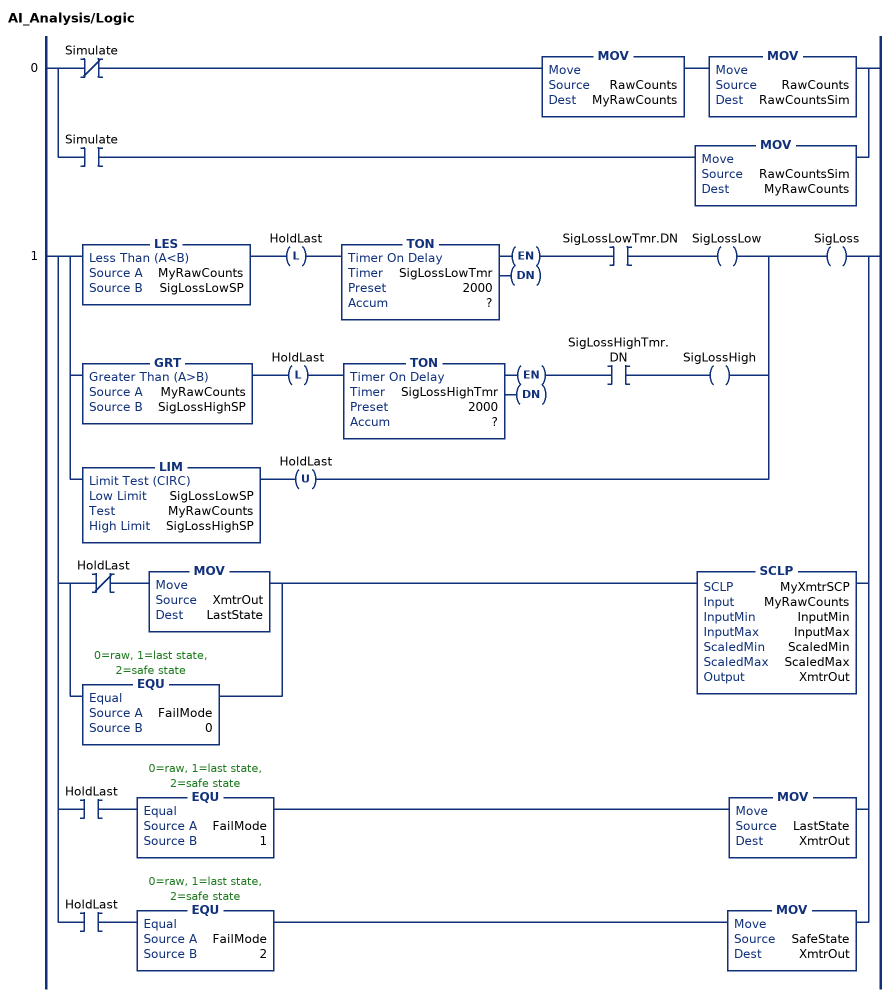
   0: [XIO(Simulate) MOV(RawCounts,MyRawCounts) MOV(RawCounts,RawCountsSim) ,XIC(Simulate) MOV(RawCountsSim,MyRawCounts) ];
   1: [[LES(MyRawCounts,SigLossLowSP) OTL(HoldLast) TON(SigLossLowTmr,?,?) XIC(SigLossLowTmr.DN) OTE(SigLossLow) ,GRT(MyRawCounts,SigLossHighSP) OTL(HoldLast) TON(SigLossHighTmr,?,?) XIC(SigLossHighTmr.DN) OTE(SigLossHigh) ,LIM(SigLossLowSP,MyRawCounts,SigLossHighSP) OTU(HoldLast) ] OTE(SigLoss) ,[XIO(HoldLast) MOV(XmtrOut,LastState) ,EQU(FailMode,0) ] SCLP(MyXmtrSCP,MyRawCounts,InputMin,InputMax,ScaledMin,ScaledMax,XmtrOut) ,XIC(HoldLast) EQU(FailMode,1) MOV(LastState,XmtrOut) ,XIC(HoldLast) EQU(FailMode,2) MOV(SafeState,XmtrOut) ];
END_ROUTINE
END_ADD_ON_INSTRUCTION

ADD_ON_INSTRUCTION AI_Compare   (* revision 1.0 *)
VAR_IN_OUT
   MyCurrentALMA : ALARM_ANALOG; {required}
   MyDefaultALMA : ALARM_ANALOG; {required}
   MyCurrentAI : AnalogControl; {required}
   MyDefaultAI : AnalogControl; {required}
END_VAR
VAR_OUTPUT
   DifferenceExists : BOOL; {access Read Only, required}
END_VAR
VAR_INPUT
   LoadDefaults : BOOL; {required}
   StoreDefaults : BOOL; {required}
END_VAR
VAR
   LimitDiff : BOOL; {access None}
   EnableDiff : BOOL; {access None}
   DeadbandDiff : BOOL; {access None}
   ROC_Diff : BOOL; {access None}
   MinDurationDiff : BOOL; {access None}
   AckRequiredDiff : BOOL; {access None}
   ScalingDiff : BOOL; {access None}
   FailModeDiff : BOOL; {access None}
END_VAR

ROUTINE Logic   (* ladder *)
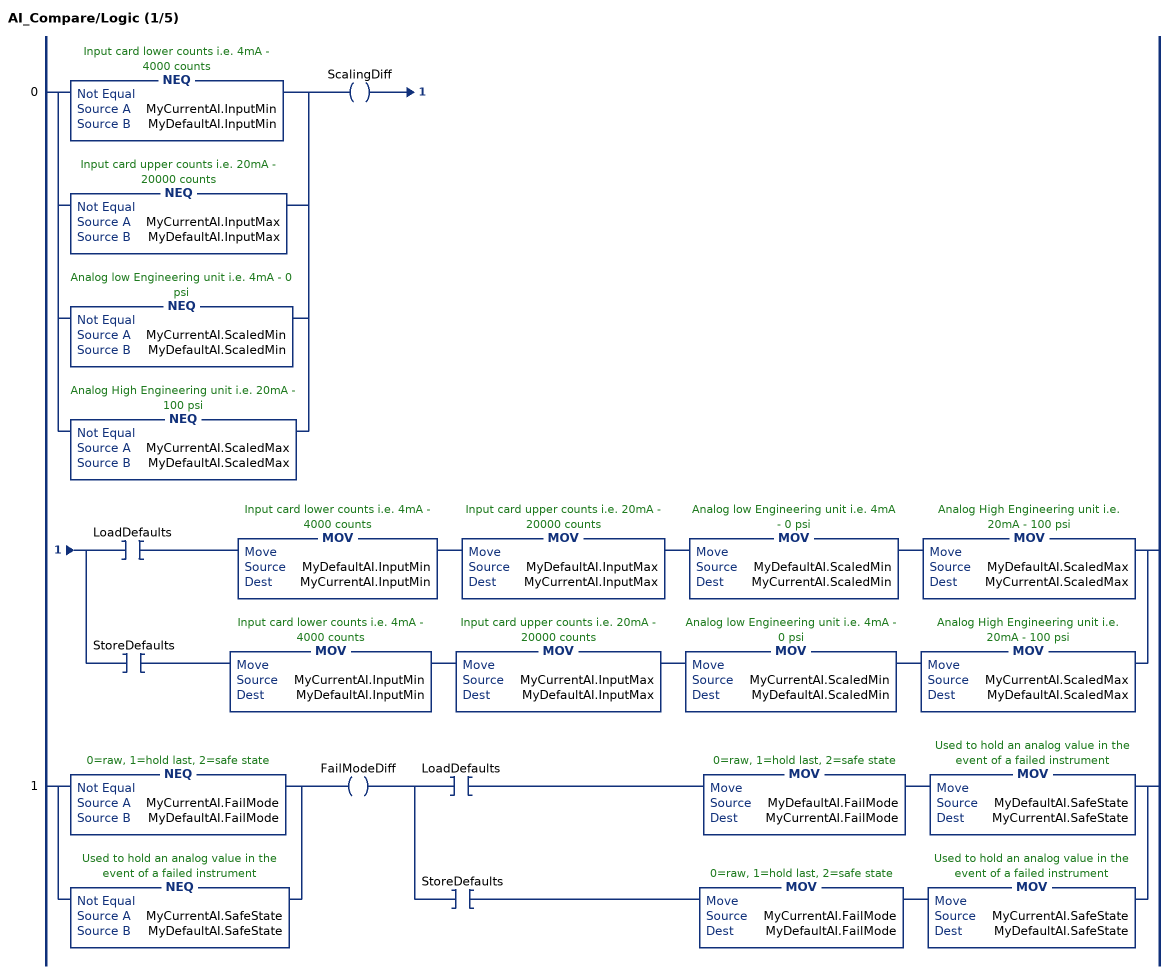
   0: [NEQ(MyCurrentAI.InputMin,MyDefaultAI.InputMin) ,NEQ(MyCurrentAI.InputMax,MyDefaultAI.InputMax) ,NEQ(MyCurrentAI.ScaledMin,MyDefaultAI.ScaledMin) ,NEQ(MyCurrentAI.ScaledMax,MyDefaultAI.ScaledMax) ]OTE(ScalingDiff)[XIC(LoadDefaults) MOV(MyDefaultAI.InputMin,MyCurrentAI.InputMin) MOV(MyDefaultAI.InputMax,MyCurrentAI.InputMax) MOV(MyDefaultAI.ScaledMin,MyCurrentAI.ScaledMin) MOV(MyDefaultAI.ScaledMax,MyCurrentAI.ScaledMax) ,XIC(StoreDefaults) MOV(MyCurrentAI.InputMin,MyDefaultAI.InputMin) MOV(MyCurrentAI.InputMax,MyDefaultAI.InputMax) MOV(MyCurrentAI.ScaledMin,MyDefaultAI.ScaledMin) MOV(MyCurrentAI.ScaledMax,MyDefaultAI.ScaledMax) ];
   1: [NEQ(MyCurrentAI.FailMode,MyDefaultAI.FailMode) ,NEQ(MyCurrentAI.SafeState,MyDefaultAI.SafeState) ]OTE(FailModeDiff)[XIC(LoadDefaults) MOV(MyDefaultAI.FailMode,MyCurrentAI.FailMode) MOV(MyDefaultAI.SafeState,MyCurrentAI.SafeState) ,XIC(StoreDefaults) MOV(MyCurrentAI.FailMode,MyDefaultAI.FailMode) MOV(MyCurrentAI.SafeState,MyDefaultAI.SafeState) ];
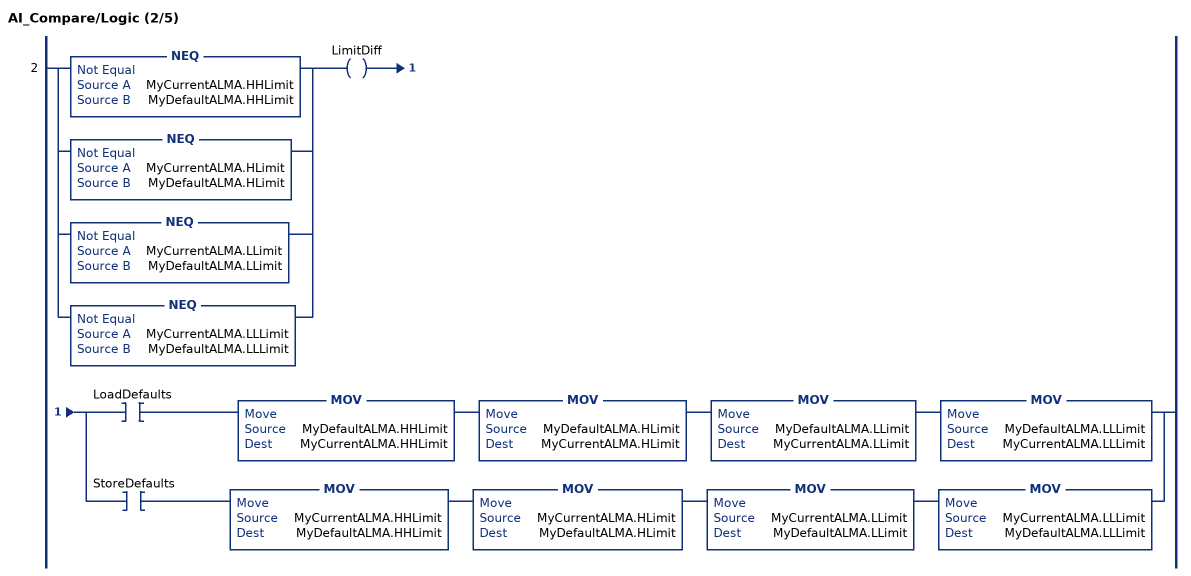
   2: [NEQ(MyCurrentALMA.HHLimit,MyDefaultALMA.HHLimit) ,NEQ(MyCurrentALMA.HLimit,MyDefaultALMA.HLimit) ,NEQ(MyCurrentALMA.LLimit,MyDefaultALMA.LLimit) ,NEQ(MyCurrentALMA.LLLimit,MyDefaultALMA.LLLimit) ]OTE(LimitDiff)[XIC(LoadDefaults) MOV(MyDefaultALMA.HHLimit,MyCurrentALMA.HHLimit) MOV(MyDefaultALMA.HLimit,MyCurrentALMA.HLimit) MOV(MyDefaultALMA.LLimit,MyCurrentALMA.LLimit) MOV(MyDefaultALMA.LLLimit,MyCurrentALMA.LLLimit) ,XIC(StoreDefaults) MOV(MyCurrentALMA.HHLimit,MyDefaultALMA.HHLimit) MOV(MyCurrentALMA.HLimit,MyDefaultALMA.HLimit) MOV(MyCurrentALMA.LLimit,MyDefaultALMA.LLimit) MOV(MyCurrentALMA.LLLimit,MyDefaultALMA.LLLimit) ];
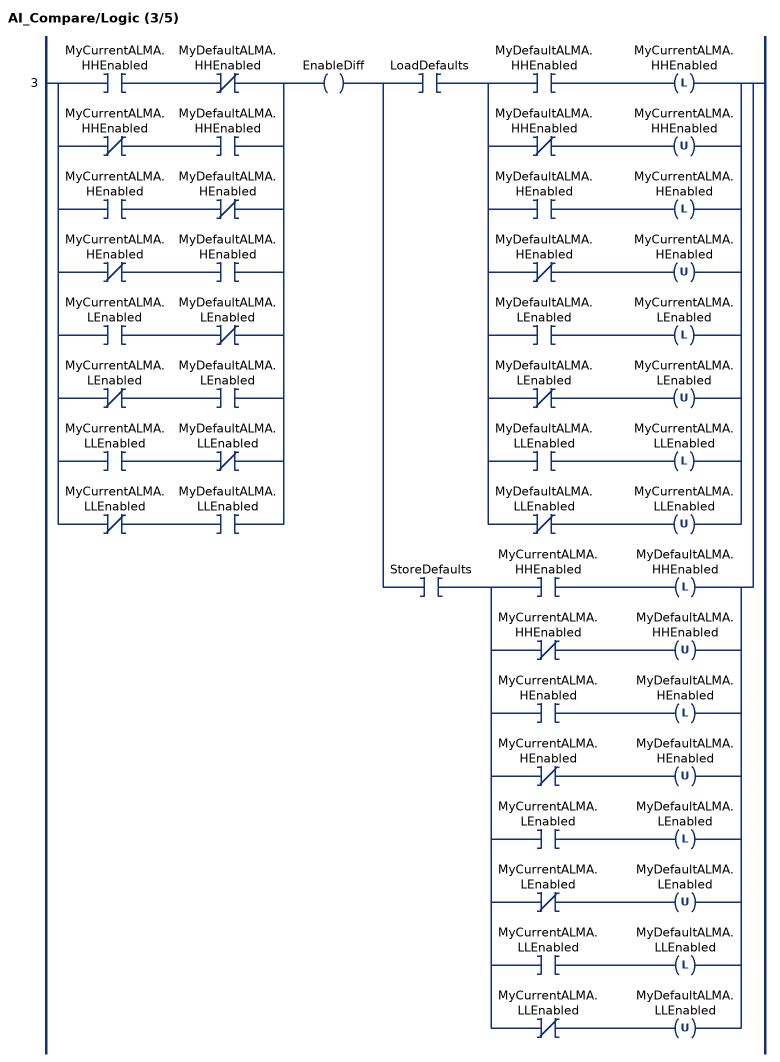
   3: [XIC(MyCurrentALMA.HHEnabled) XIO(MyDefaultALMA.HHEnabled) ,XIO(MyCurrentALMA.HHEnabled) XIC(MyDefaultALMA.HHEnabled) ,XIC(MyCurrentALMA.HEnabled) XIO(MyDefaultALMA.HEnabled) ,XIO(MyCurrentALMA.HEnabled) XIC(MyDefaultALMA.HEnabled) ,XIC(MyCurrentALMA.LEnabled) XIO(MyDefaultALMA.LEnabled) ,XIO(MyCurrentALMA.LEnabled) XIC(MyDefaultALMA.LEnabled) ,XIC(MyCurrentALMA.LLEnabled) XIO(MyDefaultALMA.LLEnabled) ,XIO(MyCurrentALMA.LLEnabled) XIC(MyDefaultALMA.LLEnabled) ]OTE(EnableDiff)[XIC(LoadDefaults) [XIC(MyDefaultALMA.HHEnabled) OTL(MyCurrentALMA.HHEnabled) ,XIO(MyDefaultALMA.HHEnabled) OTU(MyCurrentALMA.HHEnabled) ,XIC(MyDefaultALMA.HEnabled) OTL(MyCurrentALMA.HEnabled) ,XIO(MyDefaultALMA.HEnabled) OTU(MyCurrentALMA.HEnabled) ,XIC(MyDefaultALMA.LEnabled) OTL(MyCurrentALMA.LEnabled) ,XIO(MyDefaultALMA.LEnabled) OTU(MyCurrentALMA.LEnabled) ,XIC(MyDefaultALMA.LLEnabled) OTL(MyCurrentALMA.LLEnabled) ,XIO(MyDefaultALMA.LLEnabled) OTU(MyCurrentALMA.LLEnabled) ] ,XIC(StoreDefaults) [XIC(MyCurrentALMA.HHEnabled) OTL(MyDefaultALMA.HHEnabled) ,XIO(MyCurrentALMA.HHEnabled) OTU(MyDefaultALMA.HHEnabled) ,XIC(MyCurrentALMA.HEnabled) OTL(MyDefaultALMA.HEnabled) ,XIO(MyCurrentALMA.HEnabled) OTU(MyDefaultALMA.HEnabled) ,XIC(MyCurrentALMA.LEnabled) OTL(MyDefaultALMA.LEnabled) ,XIO(MyCurrentALMA.LEnabled) OTU(MyDefaultALMA.LEnabled) ,XIC(MyCurrentALMA.LLEnabled) OTL(MyDefaultALMA.LLEnabled) ,XIO(MyCurrentALMA.LLEnabled) OTU(MyDefaultALMA.LLEnabled) ] ];
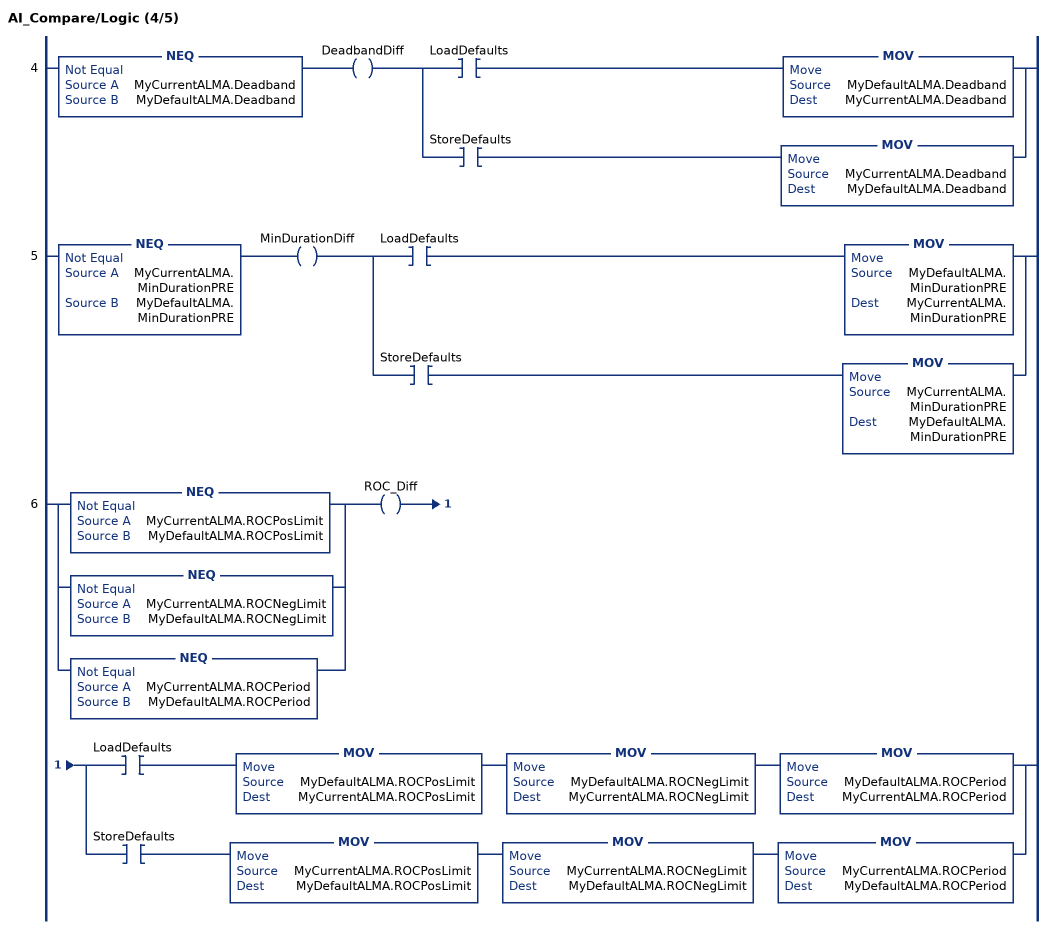
   4: NEQ(MyCurrentALMA.Deadband,MyDefaultALMA.Deadband)OTE(DeadbandDiff)[XIC(LoadDefaults) MOV(MyDefaultALMA.Deadband,MyCurrentALMA.Deadband) ,XIC(StoreDefaults) MOV(MyCurrentALMA.Deadband,MyDefaultALMA.Deadband) ];
   5: NEQ(MyCurrentALMA.MinDurationPRE,MyDefaultALMA.MinDurationPRE)OTE(MinDurationDiff)[XIC(LoadDefaults) MOV(MyDefaultALMA.MinDurationPRE,MyCurrentALMA.MinDurationPRE) ,XIC(StoreDefaults) MOV(MyCurrentALMA.MinDurationPRE,MyDefaultALMA.MinDurationPRE) ];
   6: [NEQ(MyCurrentALMA.ROCPosLimit,MyDefaultALMA.ROCPosLimit) ,NEQ(MyCurrentALMA.ROCNegLimit,MyDefaultALMA.ROCNegLimit) ,NEQ(MyCurrentALMA.ROCPeriod,MyDefaultALMA.ROCPeriod) ]OTE(ROC_Diff)[XIC(LoadDefaults) MOV(MyDefaultALMA.ROCPosLimit,MyCurrentALMA.ROCPosLimit) MOV(MyDefaultALMA.ROCNegLimit,MyCurrentALMA.ROCNegLimit) MOV(MyDefaultALMA.ROCPeriod,MyCurrentALMA.ROCPeriod) ,XIC(StoreDefaults) MOV(MyCurrentALMA.ROCPosLimit,MyDefaultALMA.ROCPosLimit) MOV(MyCurrentALMA.ROCNegLimit,MyDefaultALMA.ROCNegLimit) MOV(MyCurrentALMA.ROCPeriod,MyDefaultALMA.ROCPeriod) ];
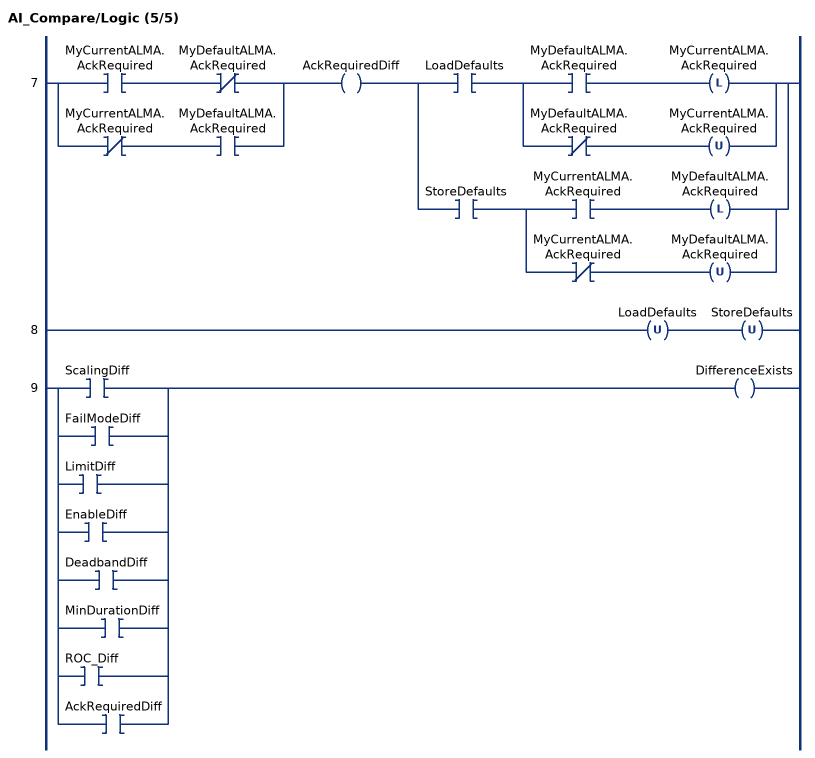
   7: [XIC(MyCurrentALMA.AckRequired) XIO(MyDefaultALMA.AckRequired) ,XIO(MyCurrentALMA.AckRequired) XIC(MyDefaultALMA.AckRequired) ]OTE(AckRequiredDiff)[XIC(LoadDefaults) [XIC(MyDefaultALMA.AckRequired) OTL(MyCurrentALMA.AckRequired) ,XIO(MyDefaultALMA.AckRequired) OTU(MyCurrentALMA.AckRequired) ] ,XIC(StoreDefaults) [XIC(MyCurrentALMA.AckRequired) OTL(MyDefaultALMA.AckRequired) ,XIO(MyCurrentALMA.AckRequired) OTU(MyDefaultALMA.AckRequired) ] ];
   8: OTU(LoadDefaults)OTU(StoreDefaults);
   9: [XIC(ScalingDiff) ,XIC(FailModeDiff) ,XIC(LimitDiff) ,XIC(EnableDiff) ,XIC(DeadbandDiff) ,XIC(MinDurationDiff) ,XIC(ROC_Diff) ,XIC(AckRequiredDiff) ]OTE(DifferenceExists);
END_ROUTINE
END_ADD_ON_INSTRUCTION

ADD_ON_INSTRUCTION AI_Simulate   (* revision 1.0 *)
VAR_INPUT
   ControlVariable : REAL; {required}
END_VAR
VAR_OUTPUT
   AI_Counts : DINT; {access Read Only, required}
END_VAR
VAR_INPUT
   RandomNumber : REAL; {required}
   PID_P : REAL; {required}
   PID_I : REAL; {required}
   ScaledMin : DINT; {required}
   ScaledMax : DINT; {required}
   Enable : BOOL; {required}
   PID_CV_Min : REAL; {required}
   PID_CV_Max : REAL; {required}
   UpdateSec : REAL; {access None, required}
   DirectActing : BOOL; {required}   // 0=Indirect (reverse) 1=Direct (forward)
END_VAR
VAR
   PID_Sim : PID := (UPD := 0.1); {access None}
   PID_Timer : TIMER := (PRE := 100); {access None}
   ProcessVariable : REAL; {access None}
   PIDControlVariable : REAL; {access None}
   SimSCLP : SCLP; {access None}
   SCLP_InputMin : REAL; {access None}
   SCLP_InputMax : REAL; {access None}
END_VAR

ROUTINE Logic   (* ladder *)
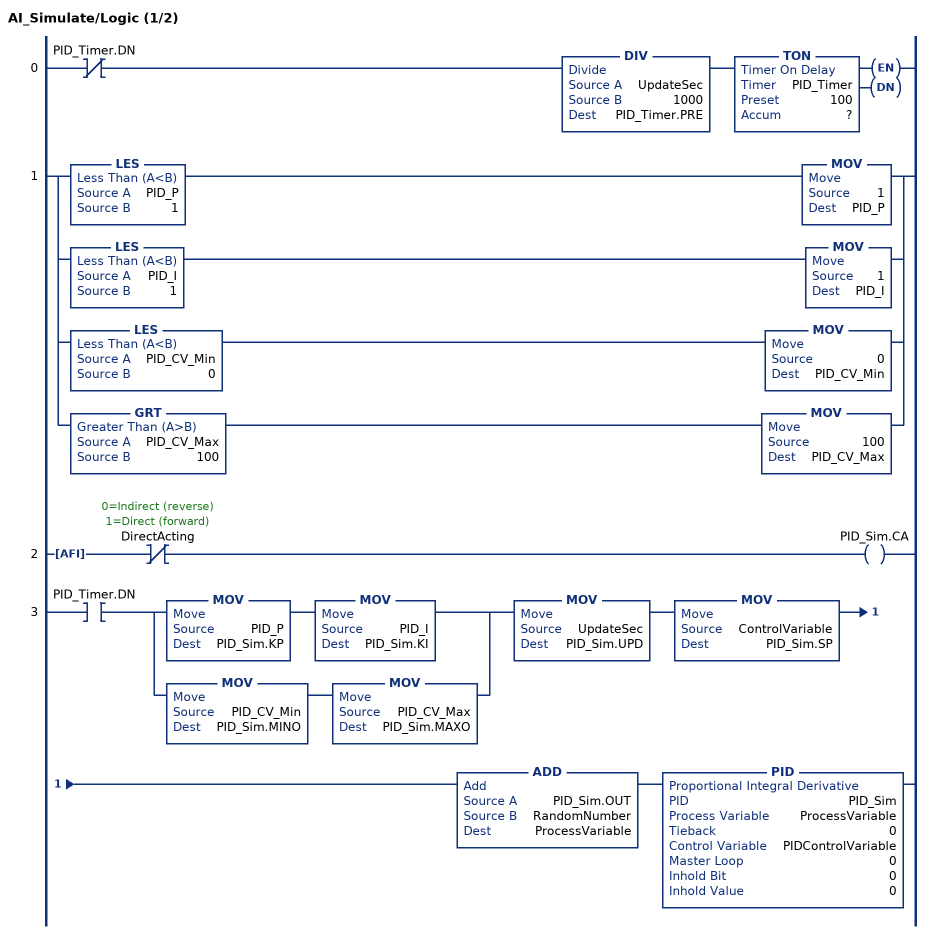
   0: XIO(PID_Timer.DN)DIV(UpdateSec,1000,PID_Timer.PRE)TON(PID_Timer,?,?);
   1: [LES(PID_P,1) MOV(1,PID_P) ,LES(PID_I,1) MOV(1,PID_I) ,LES(PID_CV_Min,0) MOV(0,PID_CV_Min) ,GRT(PID_CV_Max,100) MOV(100,PID_CV_Max) ];
   2: AFI()XIO(DirectActing)OTE(PID_Sim.CA);
   3: XIC(PID_Timer.DN)[MOV(PID_P,PID_Sim.KP) MOV(PID_I,PID_Sim.KI) ,MOV(PID_CV_Min,PID_Sim.MINO) MOV(PID_CV_Max,PID_Sim.MAXO) ]MOV(UpdateSec,PID_Sim.UPD)MOV(ControlVariable,PID_Sim.SP)ADD(PID_Sim.OUT,RandomNumber,ProcessVariable)PID(PID_Sim,ProcessVariable,0,PIDControlVariable,0,0,0);
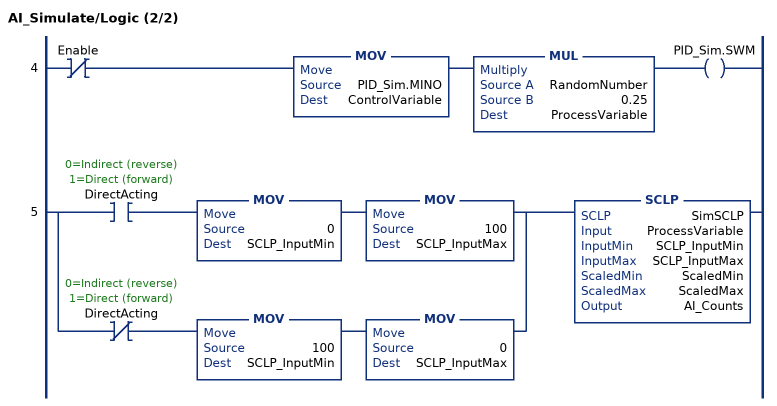
   4: XIO(Enable)MOV(PID_Sim.MINO,ControlVariable)MUL(RandomNumber,0.25,ProcessVariable)OTE(PID_Sim.SWM);
   5: [XIC(DirectActing) MOV(0,SCLP_InputMin) MOV(100,SCLP_InputMax) ,XIO(DirectActing) MOV(100,SCLP_InputMin) MOV(0,SCLP_InputMax) ]SCLP(SimSCLP,ProcessVariable,SCLP_InputMin,SCLP_InputMax,ScaledMin,ScaledMax,AI_Counts);
END_ROUTINE
END_ADD_ON_INSTRUCTION

ADD_ON_INSTRUCTION AlarmAOI   (* revision 1.0, ExecuteEnableInFalse *)
// Alarm Type
// 0 = Disabled
// 1 = Warning
// 2 = Process
// 3 = Critical
// Delay is in mSec
VAR_INPUT
   Type : DINT; {visible}   // Defines the Alarm severity. 0 = Disabled 1 = Warning 2 = Process 3 = Critical
   Override : BOOL; {required}   // Disables all Alarms
   Delay : DINT; {visible}   // Alarm Debounce in mSeconds
END_VAR
VAR_OUTPUT
   Warn : BOOL; {access Read Only, visible}   // Warning signal for HMI
   Proc : BOOL; {access Read Only, visible}   // Process signal for HMI
   Crit : BOOL; {access Read Only, visible}   // Critical Signal for HMI
END_VAR
VAR_IN_OUT
   NewAlarm : BOOL; {required}   // Requests Sonalert to turn on
   WarnExists : BOOL; {required}   // Determines if any Warnings exist
   ProcExists : BOOL; {required}   // Determines if any Process exists
   CritExists : BOOL; {required}   // Determines if any Criticals exists
END_VAR
VAR_OUTPUT
   InAlarm : BOOL; {access Read Only, visible}
END_VAR
VAR
   DelayTmr : TIMER;   // Debounce timer. Preset in mSeconds
   AlarmOffONS : BOOL;
   NewAlarmONS : BOOL;
END_VAR

ROUTINE EnableInFalse   (* ladder *)
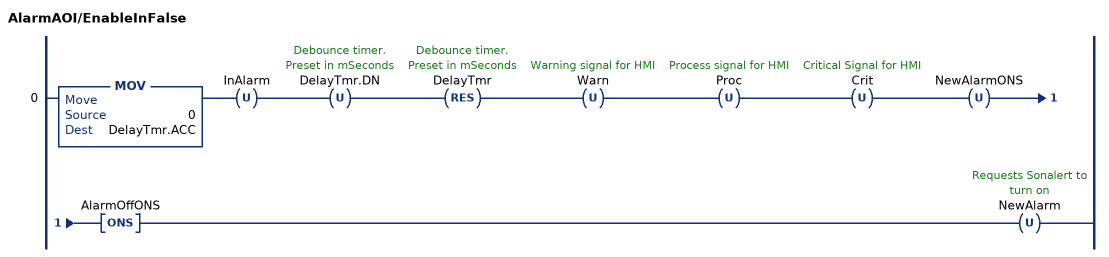
   0: MOV(0,DelayTmr.ACC)OTU(InAlarm)OTU(DelayTmr.DN)RES(DelayTmr)OTU(Warn)OTU(Proc)OTU(Crit)OTU(NewAlarmONS)ONS(AlarmOffONS)OTU(NewAlarm);
END_ROUTINE

ROUTINE Logic   (* ladder *)
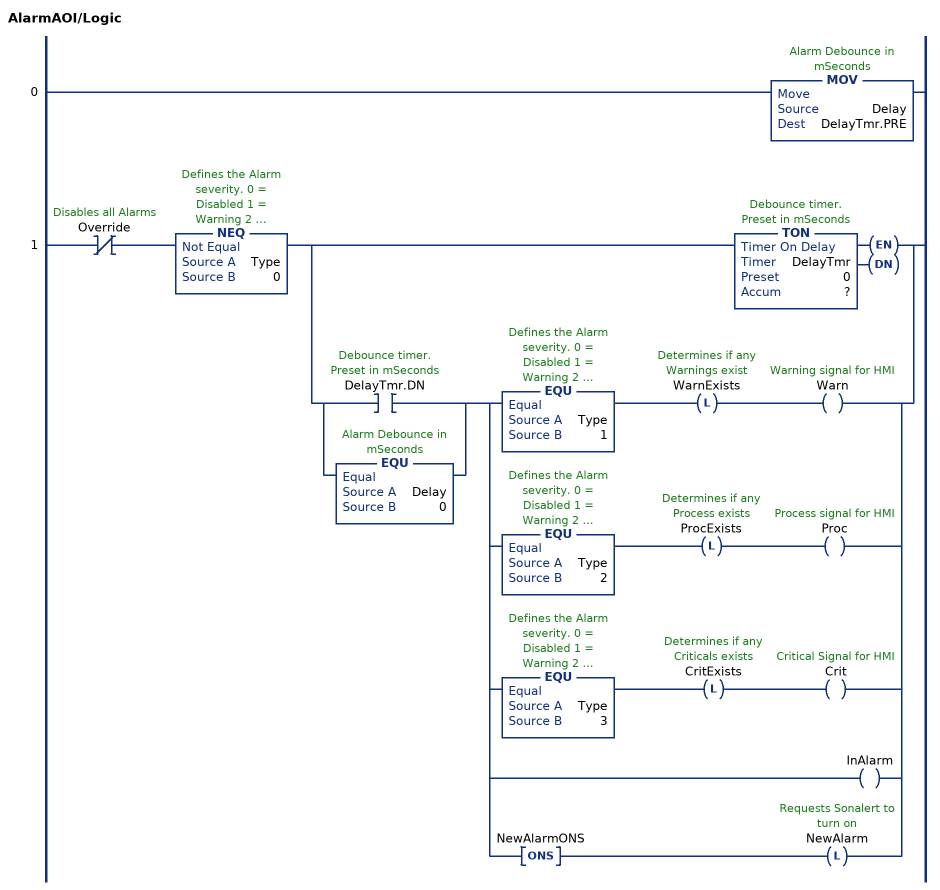
   0: MOV(Delay,DelayTmr.PRE);
   1: XIO(Override)NEQ(Type,0)[TON(DelayTmr,?,?) ,[XIC(DelayTmr.DN) ,EQU(Delay,0) ] [EQU(Type,1) OTL(WarnExists) OTE(Warn) ,EQU(Type,2) OTL(ProcExists) OTE(Proc) ,EQU(Type,3) OTL(CritExists) OTE(Crit) ,OTE(InAlarm) ,ONS(NewAlarmONS) OTL(NewAlarm) ] ];
END_ROUTINE
END_ADD_ON_INSTRUCTION

ADD_ON_INSTRUCTION MovingAve   (* revision 1.0 *)
VAR_INPUT
   InputData : REAL; {required}
   SampleRateTmrPRE : DINT; {required}
   Initialize : BOOL; {required}
   NumberOfSamples : DINT; {required}
END_VAR
VAR_IN_OUT
   OutputData : REAL; {required}
END_VAR
VAR
   MAVE_01 : MOVING_AVERAGE := (SampleEnable := 1, NumberOfSamples := 1);
   TONR_01 : FBD_TIMER;
   Storage : REAL[1000];
   MUL_01 : FBD_MATH;
   __l0000203F : BOOL; {access None}
   __l0000C226 : REAL; {access None}
   __l000018D1 : DINT; {access None}
   __l00009BB0 : DINT; {access None}
END_VAR

ROUTINE Logic   (* function block diagram *)
   SHEET 1
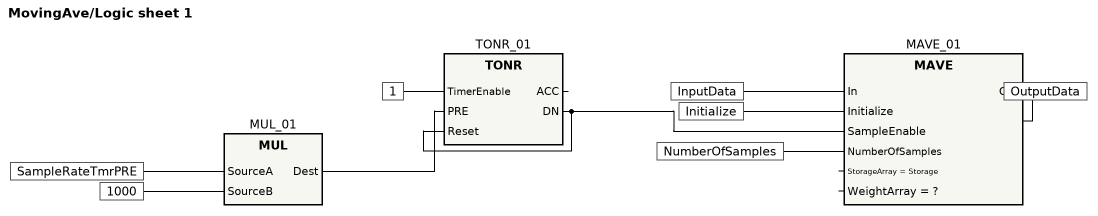
   MUL_01 : MUL(SourceA := SampleRateTmrPRE, SourceB := 1000);
   TONR_01 : TONR(TimerEnable := 1, PRE := MUL_01.Dest, Reset := TONR_01.DN);   // unwired pins: ACC
   MAVE_01 : MAVE(In := InputData, Initialize := Initialize, SampleEnable := TONR_01.DN, NumberOfSamples := NumberOfSamples, StorageArray := Storage, WeightArray := ?);
   OutputData := MAVE_01.Out;
END_ROUTINE
END_ADD_ON_INSTRUCTION

ADD_ON_INSTRUCTION PB_Toggle   (* revision 1.0, ExecuteEnableInFalse *)
// This AOI toggles a boolean tag (ie. DistPump1.Online) and resets the HMI PB.  Condition this rung with the HMI PB.
VAR_IN_OUT
   PB : BOOL; {required}
   Toggle : BOOL; {required}
END_VAR
VAR
   PBONS1 : BOOL;
   PB_Latch : BOOL;
END_VAR

ROUTINE EnableInFalse   (* ladder *)
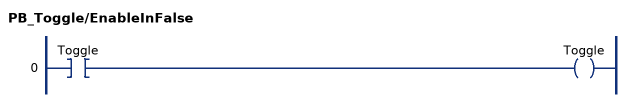
   0: XIC(Toggle)OTE(Toggle);
END_ROUTINE

ROUTINE Logic   (* ladder *)
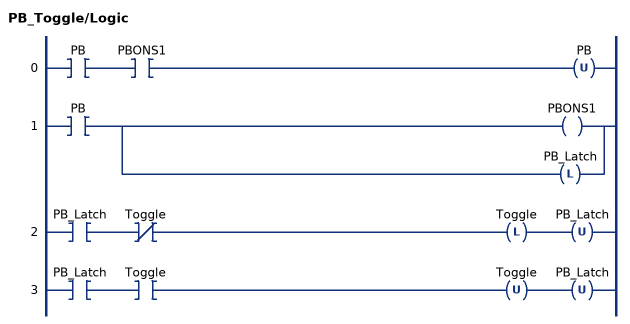
   0: XIC(PB)XIC(PBONS1)OTU(PB);
   1: XIC(PB)[OTE(PBONS1) ,OTL(PB_Latch) ];
   2: XIC(PB_Latch)XIO(Toggle)OTL(Toggle)OTU(PB_Latch);
   3: XIC(PB_Latch)XIC(Toggle)OTU(Toggle)OTU(PB_Latch);
END_ROUTINE
END_ADD_ON_INSTRUCTION

ADD_ON_INSTRUCTION SCLP   (* revision 1.0, vendor Rockwell Automation *)
VAR_INPUT
   Input : REAL; {required}
   InputMin : REAL; {required}
   InputMax : REAL; {required}
   ScaledMin : REAL; {required}
   ScaledMax : REAL; {required}
END_VAR
VAR_OUTPUT
   Output : REAL; {access Read Only, required}
END_VAR
VAR
   Temp1 : REAL;
   Temp2 : REAL;
   Rate : REAL;
   Temp4 : REAL;
   Offset : REAL;
   Temp3 : REAL;
END_VAR

ROUTINE Logic   (* ladder *)
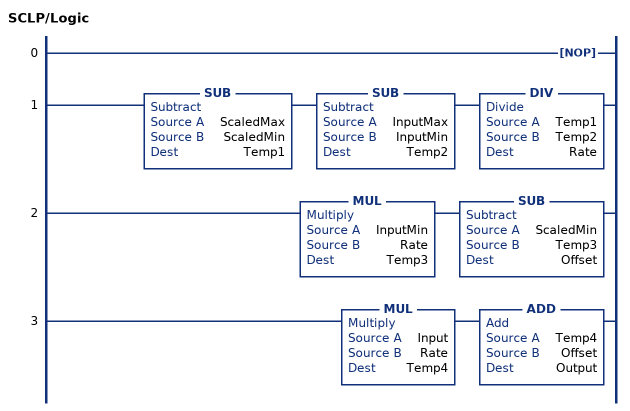
   0: NOP();
   1: SUB(ScaledMax,ScaledMin,Temp1)SUB(InputMax,InputMin,Temp2)DIV(Temp1,Temp2,Rate);
   2: MUL(InputMin,Rate,Temp3)SUB(ScaledMin,Temp3,Offset);
   3: MUL(Input,Rate,Temp4)ADD(Temp4,Offset,Output);
END_ROUTINE
END_ADD_ON_INSTRUCTION

ADD_ON_INSTRUCTION Totalize   (* revision 1.0, ExecuteEnableInFalse *)
// This instruction takes a flow signal (mL/min) and converts it to a total volume (mL)
VAR_INPUT
   FlowMeterCV : REAL; {required}
END_VAR
VAR_IN_OUT
   TotalVolume : REAL; {required}
END_VAR
VAR_INPUT
   FlowValve : BOOL; {required}
END_VAR
VAR_OUTPUT
   VolAddedLast : REAL; {access Read Only, visible}
END_VAR
VAR
   TOT_02 : TOTALIZER := (In := 2.289028, TimeBase := 1, Gain := 1.0, ProgProgReq := 1, ProgStopReq := 1, ProgResetReq := 1, OversampleDT := 0.5, RTSTime := 1, OldTotal := 413.70062, ProgOper := 1, ProgResetDone := 1, TargetFlag := 1, TargetDev1Flag := 1, TargetDev2Flag := 1, DeltaT := 0.001);
   BNOT_01 : FBD_BOOLEAN_NOT := (In := 1);
   __l0000383D : REAL; {access None}
   __l000050EC : BOOL; {access None}
END_VAR

ROUTINE EnableInFalse   (* ladder *)
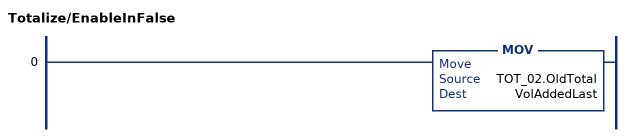
   0: MOV(TOT_02.OldTotal,VolAddedLast);
END_ROUTINE

ROUTINE Logic   (* function block diagram *)
   SHEET 1
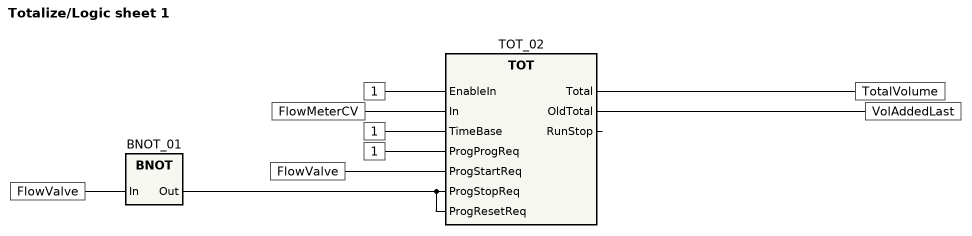
   BNOT_01 : BNOT(In := FlowValve);
   TOT_02 : TOT(EnableIn := 1, In := FlowMeterCV, TimeBase := 1, ProgProgReq := 1, ProgStartReq := FlowValve, ProgStopReq := BNOT_01.Out, ProgResetReq := BNOT_01.Out);   // unwired pins: RunStop
   TotalVolume := TOT_02.Total;
   VolAddedLast := TOT_02.OldTotal;
END_ROUTINE
END_ADD_ON_INSTRUCTION

VAR_GLOBAL   (* controller tags *)
   AC101A : ANALYTICAL := (AT := -50.0, ALL_DEV := 5.0, AL_DEV := 5.0, AH_DEV := -5.0, AHH_DEV := -5.0, AALL := 1, AAL := 1, ALL_TMR.PRE := 5000, ALL_TMR.ACC := 5000, ALL_TMR.EN := 1, ALL_TMR.DN := 1, AL_TMR.PRE := 5000, AL_TMR.ACC := 5000, AL_TMR.EN := 1, AL_TMR.DN := 1, AH_TMR.PRE := 5000, AHH_TMR.PRE := 5000, XA := 1);   // Basin Water Conductivity Control
   AC101A_SCP : SCLP := (Input := 3200.0, InputMin := 4000.0, InputMax := 20000.0, ScaledMax := 1000.0, Output := -50.0);
   AC102A : ANALYTICAL := (AUTO_SP := 70.0, CO := -0.09895, AT := -50.0, AALL_SP := 20.0, AAL_SP := 70.0, AAH_SP := 100.0, AAHH_SP := 190.0, ALL_DEV := 25.0, AL_DEV := 75.0, AH_DEV := 95.0, AHH_DEV := 185.0, ALL_TMR.PRE := 5000, AL_TMR.PRE := 5000, AH_TMR.PRE := 5000, AHH_TMR.PRE := 5000, XA := 1, RawCounts := 3200);   // QUENCH WATER CONDUCTIVITY CONTROL
   AC102A_BLEED_MAKEUP_STATUS : DINT;   // 0=stopped 1=bleed water 2=makeup water 3=wait
   AC102A_BLEED_START : BOOL;
   AC102A_BLEED_START_TON : TIMER := (PRE := 30000);
   AC102A_BLEED_STOP_TON : TIMER := (PRE := 300000);
   AC102A_BLEED_WAIT : BOOL;
   AC102A_BLEED_WAIT_TON : TIMER := (PRE := 300000);
   AC102A_MAKEUP_START : BOOL;
   AC102A_MAKEUP_STOP_TON : TIMER := (PRE := 300000);
   Alarm_New : BOOL;
   Alarm_Override : BOOL;
   Alarm_Reset : BOOL;
   AlarmMaster : DINT := 26;
        .0   // MESSAGE ALARM bit.0
        .1   // WARNING ALARM bit.1
        .2   // CSS_START_DISABLE bit.2
        .3   // PRU_START_DISABLE bit.3
        .4   // CSS_RUN_DISABLE bit.4
   AlarmMasterDisable : BOOL;
   AlarmMasterResetTON : TIMER := (PRE := 1000, ACC := 593, EN := 1, TT := 1);
   AlarmResetPB : BOOL;
   AlarmsAckAll : BOOL;
   AlarmsDisabled : BOOL;
   ALLOW : BOOL;
   AllowHeatersWhenEmpty : BOOL;
   AllowHeatersWhenEmpty_MaxMin : DINT := 1;
   AllowHeatersWhenEmpty_ONS : BOOL;
   AllowHeatersWhenEmpty_SecRemaining : DINT;
   AllowHeatersWhenEmptyONS : BOOL;
   AllowHeatersWhenEmptyTON : TIMER := (PRE := 60000);
   ALM_CRIT : BOOL;
   ALM_PROC : BOOL;
   ALM_WARN : BOOL;
   Am_I_On : BOOL := 1;
   AutoTune : PIDE_AUTOTUNE;
   BHF_TestReal : REAL := 20.0;
   bryans_gpm : REAL := 3.3;
   bryans_level : REAL := 18.9;
   Bryans_Test : BOOL;
   bryans_Test4 : BOOL;
   Bryans_Test5 : BOOL;
   bryans_test6 : BOOL;
   bryans_Test_bit : BOOL := 1;
   Bryans_Test_Int : DINT := 30;
   Bryans_Test_PID : PID := (CTL := 33612928, CA := 1, INI := 1, SPOR := 1, OLL := 1, DVNA := 1, PVHA := 1, SP := -20.0, KP := 9.867, KI := 0.1849, MAXS := 4095.0, SO := 10.0, MAXO := 40.0, MINO := 10.0, UPD := 0.5, PV := 9.368752, ERR := -15.631248, OUT := 10.0, MAXI := 4095.0, MAXCV := 100.0, MAXTIE := 4095.0, DATA[0] := 13.608395, DATA[1] := 3.6605623, DATA[2] := 9.368752, DATA[3] := -15.631248, DATA[4] := 25.0, DATA[5] := 0.024420025, DATA[6] := 1.0, DATA[7] := 8.0, DATA[8] := 9.867, DATA[9] := 0.1849, DATA[11] := 9.867, DATA[12] := 0.1849, DATA[15] := 1.0, DATA[16] := 0.024420025);
   Bryans_Test_Real : REAL;
   bryans_test_tmr : TIMER := (PRE := 1, EN := 1, TT := 1);
   Bryans_Testy_Bit : BOOL := 1;
   Coal_Tank_Heel_Inches : REAL := 16.0;
   Coal_Tank_Height_Inches : REAL := 68.0;
   ColdBoot : BOOL;
   Const_CubicInchToGal : REAL;
   CSS_Heartbeat : BOOL := 1;
   CSS_HeartbeatOffONS : BOOL;
   CSS_HeartbeatOnONS : BOOL := 1;
   CSS_HeartbeatTmr : TIMER := (PRE := 2000, ACC := 667, EN := 1, TT := 1);
   CSS_HeartbeatToggle : BOOL;
   CSS_Instrument_LOS : BOOL;   // General
   CSS_MSG_ERROR : INT;
   CSS_MSG_TMR : TIMER[16] := ([0].PRE := 10000, [1].PRE := 5000);
   CSS_OK_TO_RUN : BOOL;   // PRU_RUN_DISABLE 0 = Cannot Run 1 = OK to Run
   CSS_OK_TO_RUN_TOF : TIMER := (PRE := 10000, ACC := 10009);
   CSS_OK_TO_START : BOOL;   // PRU_START_DISABLE 0 = Cannot Start 1 = OK to Start
   CSS_OK_TO_START_TOF : TIMER := (PRE := 10000, ACC := 10000);
   CSS_REAL : REAL[100];
   CSS_STARTDISABLE : DINT;   // CSS START DISABLE
   CSS_STATUS : INT[5];
   CSS_Status_To_UTL_Comms : DINT := 9;
        .3   // PRU A IN ECOOL
        .4   // PRU B IN ECOOL
        .5   // PRU C IN ECOOL
        .6   // PRU D IN ECOOL
   DisableCommand : BOOL;
   dlm : BOOL;
   EnableCommand : BOOL;
   F1_LC302 : LEVEL_CONTROL;
   F1_LC303A : LEVEL_CONTROL;
   F1_LC370 : LEVEL_CONTROL := (AUTO_SP := 40.0);
   Fault : BOOL;
   FC101 : FLOW_CONTROL := (FT := 0.087501526, FALL_SP := 35.0, FAL_SP := 20.0, FAH_SP := 140.0, FAHH_SP := 150.0, FALL_DEV := 40.0, FAL_DEV := 25.0, FAH_DEV := 135.0, FAHH_DEV := 145.0, FALL := 1, FAL := 1, FALL_TMR.PRE := 5000, FALL_TMR.ACC := 5003, FALL_TMR.EN := 1, FALL_TMR.DN := 1, FAL_TMR.PRE := 5000, FAL_TMR.ACC := 5003, FAL_TMR.EN := 1, FAL_TMR.DN := 1, FAH_TMR.PRE := 5000, FAHH_TMR.PRE := 5000, RawCounts := 4007);   // QUENCH BASIN FLOW TRANSMITTER CONTROL
   FC101_Initialize : BOOL := 1;
   FC101_Initialize_TON : TIMER := (PRE := 1000);
   FC101_PIDE : PID_ENHANCED := (PV := 0.10000229, PVEUMax := 200.0, SPProg := -28.616238, SPCascade := -28.616238, SPHLimit := 200.0, RatioProg := 1.0, RatioOper := 1.0, RatioHLimit := 1.0, RatioLLimit := 1.0, CVEUMax := 100.0, CVHLimit := 100.0, CVLLimit := 2.0, PGain := 1.0, IGain := 5.0, PVEDerivative := 1, AllowCasRat := 1, ProgProgReq := 1, ProgManualReq := 1, RTSTime := 1, CVLAlarm := 1, SPLAlarm := 1, PVPercent := 0.050001144, E := -0.10000229, EPercent := -0.050001144, InitPrimary := 1, WindupLOut := 1, Ratio := 1.0, ProgOper := 1, Manual := 1, DeltaT := 0.01, Status1 := 16#0000_00a1, InstructFault := 1, SPProgInv := 1, SPCascadeInv := 1);
   FC108 : FLOW_CONTROL := (FT := 5.012501, FALL_SP := 15.0, FAL_SP := 21.0, FALL_DEV := 20.0, FAL_DEV := 26.0, FAH_DEV := -5.0, FAHH_DEV := -5.0, FALL := 1, FAL := 1, FAH := 1, FAHH := 1, FALL_TMR.PRE := 5000, FALL_TMR.ACC := 5014, FALL_TMR.EN := 1, FALL_TMR.DN := 1, FAL_TMR.PRE := 5000, FAL_TMR.ACC := 5013, FAL_TMR.EN := 1, FAL_TMR.DN := 1, FAH_TMR.PRE := 5000, FAH_TMR.ACC := 5001, FAH_TMR.EN := 1, FAH_TMR.DN := 1, FAHH_TMR.PRE := 5000, FAHH_TMR.ACC := 5001, FAHH_TMR.EN := 1, FAHH_TMR.DN := 1, RawCounts := 4401);   // QUENCH FEED FLOW TRANSMITTER
   FC140 : FLOW_CONTROL := (FT := -1.1499977, FALL_SP := 8.0, FAL_SP := 10.0, FAH_SP := 1.0, FAHH_SP := 25.0, FALL_DEV := 6.0, FAL_DEV := 8.0, FAH_DEV := -1.0, FAHH_DEV := 23.0, FALL_TMR.PRE := 5000, FAL_TMR.PRE := 5000, FAH_TMR.PRE := 5000, FAHH_TMR.PRE := 5000, Simulate := 1);
   FC140_DIFF_FT : REAL := 1.25;
   FC140A : FLOW_CONTROL := (FT := 0.10000229, FALL_SP := 10.0, FAL_SP := 16.0, FAH_SP := 190.0, FAHH_SP := 200.0, FALL_DEV := 12.0, FAL_DEV := 18.0, FAH_DEV := 188.0, FAHH_DEV := 198.0, FALL := 1, FAL := 1, FALL_TMR.PRE := 20000, FALL_TMR.ACC := 20008, FALL_TMR.EN := 1, FALL_TMR.DN := 1, FAL_TMR.PRE := 20000, FAL_TMR.ACC := 20010, FAL_TMR.EN := 1, FAL_TMR.DN := 1, FAH_TMR.PRE := 5000, FAHH_TMR.PRE := 5000, RawCounts := 4008);   // QUENCH TOWER UPPER SPRAY FLOW CONTROL
   FC140A_FT_Pcnt : REAL := 0.07407565;
   FC140A_FT_Percent : DINT;
   FC140B : FLOW_CONTROL := (FT := 1.25, FALL_SP := 10.0, FAL_SP := 20.0, FAH_SP := 190.0, FAHH_SP := 200.0, FALL_DEV := 12.0, FAL_DEV := 22.0, FAH_DEV := 188.0, FAHH_DEV := 198.0, FALL := 1, FAL := 1, FALL_TMR.PRE := 20000, FALL_TMR.ACC := 20006, FALL_TMR.EN := 1, FALL_TMR.DN := 1, FAL_TMR.PRE := 20000, FAL_TMR.ACC := 20008, FAL_TMR.EN := 1, FAL_TMR.DN := 1, FAH_TMR.PRE := 5000, FAHH_TMR.PRE := 5000, RawCounts := 4100);   // QUENCH TOWER LOWER SPRAY FLOW CONTROL
   FC140B_FT_Pcnt : REAL := 0.92592436;
   FC141 : PUMP_CONTROL;
   FC215 : FLOW_CONTROL := (FT := 0.018751144, FALL_DEV := 5.0, FAL_DEV := 5.0, FAH_DEV := -5.0, FAHH_DEV := -5.0, FALL := 1, FAL := 1, FAH := 1, FAHH := 1, FALL_TMR.PRE := 5000, FALL_TMR.ACC := 5011, FALL_TMR.EN := 1, FALL_TMR.DN := 1, FAL_TMR.PRE := 5000, FAL_TMR.ACC := 5011, FAL_TMR.EN := 1, FAL_TMR.DN := 1, FAH_TMR.PRE := 5000, FAH_TMR.ACC := 5000, FAH_TMR.EN := 1, FAH_TMR.DN := 1, FAHH_TMR.PRE := 5000, FAHH_TMR.ACC := 5000, FAHH_TMR.EN := 1, FAHH_TMR.DN := 1, RawCounts := 4004);   // OVERHEAD CONDENSER CHILLED WATER FLOW CONTROL
   FC365 : FLOW_CONTROL := (AUTO := 1, AUTO_SP := 70.0, FT := 0.0015624762, FALL_SP := 0.5, FAL_SP := 1.0, FAH_SP := 4.0, FAHH_SP := 4.8, FALL_DEV := 0.75, FAL_DEV := 1.25, FAH_DEV := 3.75, FAHH_DEV := 4.55, FALL_TMR.PRE := 5000, FAL_TMR.PRE := 5000, FAH_TMR.PRE := 5000, FAHH_TMR.PRE := 5000, RawCounts := 4005, AI_Anal.XmtrOut := 0.0015624762, AI_Anal.RawCounts := 4005, AI_Anal.SigLossHighSP := 21000, AI_Anal.SigLossLowSP := 3810, AI_Anal.InputMin := 4000.0, AI_Anal.InputMax := 20000.0, AI_Anal.ScaledMax := 5.0, AI_Anal.RawCountsSim := 4005, InputMin := 4000, InputMax := 20000, ScaledMax := 5.0, PV := 0.0015624762);   // COALESCER PROCESS IMPURITY FLOW CONTROL
   FC365_AI_Compare : AI_Compare;
   FC365_Alm : ALARM_ANALOG;
   FC365_AlmDefault : ALARM_ANALOG;
   FC365_AUTO_ONS1 : BOOL := 1;
   FC365_AUTO_ONS2 : BOOL;
   FC365_BLEED_ALARM_DISABLE : BOOL := 1;
   FC365_BLEED_FLOW_MIN_SP : DINT := 5;
   FC365_BLEED_WAIT_MIN_SP : DINT := 5;
   FC365_FLOW_TOO_LONG_ALM : BOOL;
   FC365_FLOW_TOO_LONG_RESETPB : BOOL;
   FC365_FLOW_TOO_LONG_TMR : TIMER := (PRE := 1800000);
   FC365_HMI_BLEED_REQ : BOOL;
   FC365_HMI_BLEED_REQ_ONS : BOOL;
   FC365_HMI_BLEED_START_ENABLE : BOOL;
   FC365_HMI_BLEED_START_ENABLE_TON : TIMER := (PRE := 30000);
   FC365_HMI_BLEED_START_PB : BOOL;
   FC365_HMI_BLEED_STOP_PB : BOOL;
   FC365_HMI_VERIFY_PB : BOOL;
   FC365_LC370_FLOW_AUTO_SP : REAL := 3.0;
   FC365_MANUAL_ONS1 : BOOL;
   FC365_MAX_TIME_MIN : DINT := 30;
   FC365_Started : BOOL;
   FC365_TOTAl_GAL : REAL := 43009.156;
   FC365_TOTAl_RESET : BOOL := 1;
   FC365_TOTAl_RESET_PB : BOOL;
   FC365_TOTALIZE : Totalize := (FlowMeterCV := 0.0012500286, FlowValve := 1, VolAddedLast := 4965.832);
   FC365_TOTALIZE_EN : BOOL;
   FC365_TOTALIZE_EN_ONS1 : BOOL := 1;
   FC365_TOTALIZE_GPM : REAL;
   FC365_TOTALIZE_LastFeedTimeMin : REAL := 166.66678;
   FC365_TOTALIZE_Min : REAL := 166.66678;
   FC365_TOTALIZE_TON : TIMER := (PRE := 9999999);
   FC365_UNABLE_TO_BLEED : BOOL;
   FC370 : FLOW_CONTROL := (MAN_SP := 61.434135, CO := 70.0, FT := -0.0006250143, FALL_DEV := 5.0, FAL_DEV := 5.0, FAH_DEV := -5.0, FAHH_DEV := -5.0, FALL_TMR.PRE := 5000, FAL_TMR.PRE := 5000, FAH_TMR.PRE := 5000, FAHH_TMR.PRE := 5000, RawCounts := 3998);   // COALESCER MAKE UP WATER FLOW CONTROL
   FC370_FEED_ALARM_DISABLE : BOOL := 1;
   FC370_Open : BOOL;
   FC370_Totalize : Totalize;
   FC370_TotalVolume : REAL;
   FC403 : FLOW_CONTROL := (FT := 0.10000229, FALL_SP := 100.0, FAL_SP := 110.0, FAH_SP := 220.0, FAHH_SP := 230.0, FALL_DEV := 105.0, FAL_DEV := 115.0, FAH_DEV := 215.0, FAHH_DEV := 225.0, FALL := 1, FAL := 1, FALL_TMR.PRE := 5000, FALL_TMR.ACC := 5003, FALL_TMR.EN := 1, FALL_TMR.DN := 1, FAL_TMR.PRE := 5000, FAL_TMR.ACC := 5003, FAL_TMR.EN := 1, FAL_TMR.DN := 1, FAH_TMR.PRE := 5000, FAHH_TMR.PRE := 5000, RawCounts := 4008);   // COALESCER FLOW CONTROLLER FEEDS TCV108
   FC406 : FLOW_CONTROL := (AUTO := 1, MAN_SP := 100.0, FT := 0.03750229, FALL_DEV := 5.0, FAL_DEV := 5.0, FAH_DEV := -5.0, FAHH_DEV := -5.0, FALL := 1, FAL := 1, FAH := 1, FAHH := 1, FALL_TMR.PRE := 5000, FALL_TMR.ACC := 5010, FALL_TMR.EN := 1, FALL_TMR.DN := 1, FAL_TMR.PRE := 5000, FAL_TMR.ACC := 5010, FAL_TMR.EN := 1, FAL_TMR.DN := 1, FAH_TMR.PRE := 5000, FAH_TMR.ACC := 5006, FAH_TMR.EN := 1, FAH_TMR.DN := 1, FAHH_TMR.PRE := 5000, FAHH_TMR.ACC := 5007, FAHH_TMR.EN := 1, FAHH_TMR.DN := 1, RawCounts := 4003);   // HX COOLING WATER FLOW CONTROL
   FC_215 : FLOW_CONTROL := (FT := 40.9);
   FC_215SCP : SCLP := (Input := 4004.0, InputMin := 4000.0, InputMax := 20000.0, ScaledMax := 75.0, Output := 0.018751144);   // OVERHEAD CONDENSER CHILLED WATER FLOW TRANSMITTER SCALER
   FC_406 : FLOW_CONTROL := (FT := 0.04999);
   FC_406SCP : SCLP := (Input := 4004.0, InputMin := 4000.0, InputMax := 20000.0, ScaledMax := 200.0, Output := 0.049999237);   // HX COOLING WATER FLOW TRANMITTER SCALER
   FCV141_AUTO_ONS : BOOL;
   FCV141_MANUAL_ONS : BOOL;
   FCV141_MaxOpenSecSP : REAL := 6.0;
   FCV141_MaxOpenTmr : TIMER := (PRE := 6000);
   FCV141_Open : BOOL;
   FCV365_SCLP : SCLP := (InputMax := 100.0, ScaledMin := 4000.0, ScaledMax := 20000.0, Output := 4000.0);   // SEPARATOR PROCESS IMPURITY BLEED CONTROL OUTPUT SCALER
   FCV365_SCP : SCLP := (Input := 3200.0, InputMin := 4000.0, InputMax := 20000.0, ScaledMax := 100.0, Output := -5.0);
   FCV410 : ValveControl_TwoWay := (Auto := 1);
   FCV410_AUTO_ONS : BOOL := 1;
   FCV410_ClosedMinSP : DINT := 15;
   FCV410_ClosedTON : TIMER := (PRE := 900000, ACC := 316117, EN := 1, TT := 1);
   FCV410_HoldDelaySecSP : DINT := 15;
   FCV410_HoldDelayTOF : TIMER := (PRE := 15000, ACC := 15006);
   FCV410_LT_Hold : BOOL;
   FCV410_MANUAL_ONS : BOOL;
   FCV410_On : BOOL;
   FCV410_Open : BOOL;
   FCV410_OpenSecSP : DINT := 10;
   FCV410_OpenTON : TIMER := (PRE := 10000);
   FireFlowAlarm_ONS1 : BOOL;
   FireFlowAlarm_ONS2 : BOOL := 1;
   FireFlowAlarm_SetLC101 : BOOL := 1;
   FireFlowAlarmFromUTL : BOOL := 1;
   FireFlowAlarmLC101_SP : REAL := 10.0;
   FireFlowLC370_SP : REAL := 45.0;
   FirstScanLatch : BOOL;
   FirstScanLatchTON : TIMER := (PRE := 20000);
   FIT08 : BOOL := 1;
   FIT101 : BOOL := 1;
   FIT140A : BOOL := 1;
   FIT140B : BOOL := 1;
   FIT365 : REAL;
   FIT365_SCP : SCLP := (Input := 4005.0, InputMin := 4000.0, InputMax := 20000.0, ScaledMax := 5.0, Output := 0.0015624762);   // COALESCER PROCESS IMPURITY FLOW
   FIT370_SCP : SCLP := (Input := 3999.0, InputMin := 4000.0, InputMax := 20000.0, ScaledMax := 5.0, Output := -0.00031256676);   // COALESCER MAKE UP WATER SCALER
   FIT403 : BOOL := 1;
   FlowControlForce : BOOL;
   FlowControlForceONS : BOOL;
   FQT365 : REAL;
   FT101 : REAL := 15.275002;   // QUENCH TOWER BASIN FLOW
   FT101_SCP : SCLP := (Input := 4008.0, InputMin := 4000.0, InputMax := 20000.0, ScaledMax := 200.0, Output := 0.10000229);   // QUENCH BASIN FLOW TRANSMITTER SCALER
   FT108 : REAL := 67.4125;   // QUENCH TOWER GAS FRACTION FLOW
   FT108_SCP : SCLP := (Input := 4403.0, InputMin := 4000.0, InputMax := 20000.0, ScaledMax := 200.0, Output := 5.0375023);   // QUENCH FEED FLOW TRANSMITTER SCALER
   FT140_Ratio : REAL := 1.3500023;
   FT140_TOTAL : DINT := 70;
   FT140_TOTAL_FLOW : REAL := 1.3500023;
   FT140A : REAL := 38.012505;   // QUENCH TOWER UPPER SPRAY FIT
   FT140A_SCP : SCLP := (Input := 4008.0, InputMin := 4000.0, InputMax := 20000.0, ScaledMax := 200.0, Output := 0.10000229);   // QUENCH TOWER UPPER SPRAY FIT SCALER
   FT140ABFlowMeterFailed : BOOL;
   FT140B : REAL := 74.4875;   // QUENCH TOWER LOWER SPRAY
   FT140B_SCP : SCLP := (Input := 4100.0, InputMin := 4000.0, InputMax := 20000.0, ScaledMax := 200.0, Output := 1.25);   // QUENCH TOWER LOWER SPRAY FLOW TRANSMITTER SCALER
   FT403 : REAL := 67.22813;   // QUENCH CONDITIONING QUENCH WATER PHASE FLOW SCALER
   FT403_SCP : SCLP := (Input := 4008.0, InputMin := 4000.0, InputMax := 20000.0, ScaledMax := 200.0, Output := 0.10000229);   // QUENCH CONDITIONING QUENCH WATER PHASE FLOW SCALER
   GTL_TDAHH_MinSP : REAL := 400.0;
   H3_LC101 : LEVEL_CONTROL := (AUTO_SP := 10.0);
   HART1 : HARTModuleDef := (GenStat.Scan_Cnt := 1006, GenStat.Product_Name[0] := 72, GenStat.Product_Name[1] := 82, GenStat.Product_Name[2] := 84, GenStat.Product_Name[3] := 54, GenStat.Rev_Level[0] := 50, GenStat.Rev_Level[1] := 46, GenStat.Rev_Level[2] := 48, GenStat.Rev_Level[3] := 52, GenStat.Op_Sys[0] := 48, GenStat.Op_Sys[1] := 55, GenStat.Op_Sys[2] := 48, GenStat.Op_Sys[3] := 52, GenStat.Run_Number[0] := 48, GenStat.Run_Number[1] := 55, GenStat.Run_Number[2] := 48, GenStat.Run_Number[3] := 49, GenStat.Blk_Rd_Count := 31730, GenStat.Blk_Wr_Count := 31731, GenStat.Blk_Parse_Cnt := 31731, GenStat.Blk_Err := 758, GenStat.ChStat[0].State := 3, GenStat.ChStat[0].Comm_State := 6, GenStat.ChStat[0].Dev_in_poll := 2#0000_0000_0000_0100, GenStat.ChStat[0].Dev_long := 2#0000_0000_0000_0100, GenStat.ChStat[0].Cur_cmd := 1, GenStat.ChStat[0].Cmd_req := 10871, GenStat.ChStat[0].Cmd_resp := 10860, GenStat.ChStat[0].LastErr := 64, GenStat.ChStat[1].Comm_State := 6, GenStat.ChStat[1].Dev_stat := 2#0000_0000_0011_1110, GenStat.ChStat[1].Dev_in_poll := 2#0000_0000_0011_1110, GenStat.ChStat[1].Cmd_req := 13573, GenStat.ChStat[1].CurErr := -1, BP.LastRead := 3, BP.LastWrite := 4, BP.BlockIndex := 360, Auto_Poll[0].Secondary_Var_Units := -68, Auto_Poll[0].Tertiary_Var_Units := 3, Auto_Poll[0].Quaternary_Var_Units := 72, Auto_Poll[0].Tag_Name[0] := 'R', Auto_Poll[0].Tag_Name[1] := 'T', Auto_Poll[0].Tag_Name[2] := '6', Auto_Poll[0].Tag_Name[3] := '2', Auto_Poll[0].Tag_Name[4] := '.', Auto_Poll[0].Tag_Name[5] := '0', Auto_Poll[0].Tag_Name[6] := '4', Auto_Poll[0].Tag_Name[7] := '0', Auto_Poll[0].Descriptor[0] := '7', Auto_Poll[0].Descriptor[1] := '0', Auto_Poll[0].Descriptor[2] := '4', Auto_Poll[0].Descriptor[3] := '0', Auto_Poll[0].Descriptor[4] := '7', Auto_Poll[0].Descriptor[5] := '0', Auto_Poll[0].Descriptor[6] := '1', Auto_Poll[0].Descriptor[7] := '$F0', Auto_Poll[0].Descriptor[8] := '{', Auto_Poll[0].Descriptor[9] := '$F0', Auto_Poll[0].Descriptor[10] := '{', Auto_Poll[0].Descriptor[11] := '$F0',
        Auto_Poll[0].Descriptor[12] := '{', Auto_Poll[0].Tag_Descriptor_Data[1] := '$F6', Auto_Poll[0].Tag_Descriptor_Data[2] := '$02', Auto_Poll[0].Transd_Serial_Num[0] := 3, Auto_Poll[0].Transd_Serial_Num[2] := 6, Auto_Poll[0].PV_URLLRV_Units := 4, Auto_Poll[0].Private_Label_Code := 4, Auto_Poll[0].PV_value := 2.1938008e-13, Auto_Poll[0].SV_value := 1.5218e-41, Auto_Poll[0].TV_value := 5.877472e-39, Auto_Poll[0].QV_value := 4.59177e-40, Auto_Poll[0].U_trans_limit := 5.693888e-39, Auto_Poll[0].Min_span := 1.9018e-41, Auto_Poll[0].PV_URV := nan, BlockTransferSize := 120);
        .GENSTAT.SCAN_CNT   // This should always be counting, always changing. If not then lost coms with processor or locked up
        .GENSTAT.PRODUCT_NAME   // should be set up as ascii
        .GENSTAT.REV_LEVEL   // should be set up as ascii
        .GENSTAT.BLK_RD_COUNT   // these both should be continually counting
        .GENSTAT.BLK_WR_COUNT   // these both should be continually counting
        .GENSTAT.CHSTAT[0].COMM_STATE   // should be moving between 1 and 6 post transmit, idle
        .GENSTAT.CHSTAT[0].STATE   // user poll "3" command
        .GENSTAT.CHSTAT[0].CMD_RESP   // replies
        .GENSTAT.CHSTAT[0].CMD_REQ   // count of sending responses
   HART_CH1 : REAL[10];
   HART_CH2 : REAL[10];
   HARTData1 : HARTData := (HART_IN_Int_vals[10] := 956, HART_IN_Int_vals[11] := 21064, HART_IN_Int_vals[12] := 13908, HART_IN_Int_vals[13] := 11826, HART_IN_Int_vals[14] := 13360, HART_IN_Int_vals[15] := 14128, HART_IN_Int_vals[16] := 13360, HART_IN_Int_vals[17] := 14128, HART_IN_Int_vals[18] := 12592, HART_IN_Int_vals[19] := 31728, HART_IN_Int_vals[20] := 31728, HART_IN_Int_vals[21] := 31728, HART_IN_Int_vals[24] := 758, HART_IN_Int_vals[25] := 3, HART_IN_Int_vals[26] := 6, HART_IN_Int_vals[28] := 4, HART_IN_Int_vals[29] := 4, HART_IN_Int_vals[30] := 1, HART_IN_Int_vals[31] := 10871, HART_IN_Int_vals[32] := 10860, HART_IN_Int_vals[35] := 64, HART_IN_Int_vals[37] := 5, HART_IN_Int_vals[38] := 62, HART_IN_Int_vals[39] := 62, HART_IN_Int_vals[42] := 13572, HART_IN_Int_vals[45] := -1, HART_IN_Int_vals[90] := 62, HART_IN_Int_vals[100] := -15556, HART_IN_Int_vals[101] := 16546, HART_IN_Int_vals[102] := 17463, HART_IN_Int_vals[103] := 16601, HART_IN_Int_vals[104] := 17463, HART_IN_Int_vals[105] := 16601, HART_IN_Int_vals[108] := 24499, HART_IN_Int_vals[109] := 17222, HART_IN_Int_vals[110] := 16384, HART_IN_Int_vals[111] := 14649, HART_IN_Int_vals[112] := 9273);
   HCP_FAULT : BOOL := 1;
   HEART_DATA : INT[122] := ([0] := 4);
   HeaterControl_IgnoreLevel : BOOL;
   HeaterControl_IgnoreLevel_ONS : BOOL;
   HeaterControl_IgnoreLevelSecSP : DINT;
   HeaterControl_IgnoreLevelTMR : TIMER;
   HMI_ShowReboot : BOOL;
   HMI_ShowRebootTmr : TIMER := (PRE := 5000);
   HS104A : ValveControl_TwoWay := (Manual := 1, Auto := 1);
   HS104B : ValveControl_TwoWay := (Manual := 1, Auto := 1);
   HS141 : ValveControl_TwoWay;
   HS315A : ValveControl_TwoWay := (Manual := 1, Auto := 1);
   HS315A_AUTO_ONS : BOOL;
   HS315A_Energized : BOOL;
   HS315A_MANUAL_ONS : BOOL;
   HS315B : ValveControl_TwoWay := (Manual := 1, Auto := 1);
   HS431A : ValveControl_TwoWay := (Status := 1, Auto := 1);
   HS431B : ValveControl_TwoWay := (Status := 1, Auto := 1);
   HS433A : ValveControl_TwoWay := (Status := 1, Auto := 1);
   HS433B : ValveControl_TwoWay := (Status := 1, Auto := 1);
   HT_FAULT : BOOL;
   HTGA : BOOL;
   HX401_TRANSFER_LEAD_TON : TIMER := (PRE := 3600000, ACC := 1545591, EN := 1, TT := 1);
   HX401A : PUMP_CONTROL := (QI_AUTO := 1, QI_LEAD := 1, QI_TRANSFER_LEAD := 1, START := 1, LEAD_DAYS_SP := 2, LEAD_XFER_TMR.PRE := 5000, RUN_HRS.PRE := 7200000, RUN_HRS.ACC := 7200000, RUN_HRS.EN := 1, RUN_HRS.DN := 1, START_DELAY.PRE := 1000, START_DELAY.ACC := 1005, START_DELAY.EN := 1, START_DELAY.DN := 1);   // HEAT EXCHANGER A
   HX401A_QI_AUTO_OS : BOOL := 1;
   HX401A_QI_MAN_OS : BOOL;
   HX401B : PUMP_CONTROL := (QI_MANUAL := 1, QI_TRANSFER_LEAD := 1, QI_RUN_STATUS := 1, START := 1, LEAD_DAYS_SP := 1, LEAD_XFER_TMR.PRE := 5000, RUN_HRS.PRE := 3600000, RUN_HRS.ACC := 3600008, RUN_HRS.EN := 1, RUN_HRS.DN := 1, START_DELAY.PRE := 1000, START_DELAY.ACC := 1005, START_DELAY.EN := 1, START_DELAY.DN := 1);   // HEAT EXCHANGER B
   HX401B_QI_AUTO_OS : BOOL;
   HX401B_QI_MAN_OS : BOOL := 1;
   HX431B_OPEN : BOOL;   // H431B HX B VALVE OPEN FAIL OPEN ENERGIZE TO CLOSE
   InputMax_IF8 : REAL := 20000.0;
   InputMin_IF8 : REAL := 4000.0;
   Instrument_LOS : BOOL[32] := ([0] := 1, [1] := 1, [2] := 1);
   IP_Address : DINT[4] := ([0] := 192, [1] := 168, [2] := 20, [3] := 70);
   IP_AddressGetMSG : MESSAGE;
        MessageParameters(ServiceCode := 16#000e, DestinationTag := TCP_GetAll, ...)
   IP_AddressGetMSG_TON : TIMER := (PRE := 10000, ACC := 3215, EN := 1, TT := 1);
   IP_AddressSetMSG : MESSAGE;
        MessageParameters(ServiceCode := 16#0010, LocalElement := TCP_SetAll, ...)
   IsThisOn : DINT := 3;
   JC102_SCLP : SCLP := (InputMax := 100.0, ScaledMin := 4000.0, ScaledMax := 20000.0, Output := 4000.0);
   JC114_SCLP : SCLP := (InputMax := 100.0, ScaledMin := 4000.0, ScaledMax := 20000.0, Output := 4000.0);   // QUENCH BASIN HEAT CONTROLLE CONTROL OUTPUT SCALER
   JC306_SCLP : SCLP := (InputMax := 100.0, ScaledMin := 4000.0, ScaledMax := 20000.0, Output := 4000.0);   // OIL TRANSFER CHAMBER HEAT CONTROLLER CONTROL OUTPUT SCALER
   JC313A_SCLP : SCLP := (InputMax := 100.0, ScaledMin := 4000.0, ScaledMax := 20000.0, Output := 4000.0);   // PRIMARY SETTLER HEAT CONTROLLER CONTROL OUTPUT SCALER
   LC101 : LEVEL_CONTROL := (AUTO := 1, AUTO_SP := 20.0, CO := 100.0, FB := 100.0, PID_CO := 5.0, LT := 42.0985, LALL_SP := 10.0, LAL_SP := 15.0, LAH_SP := 24.0, LAHH_SP := 28.0, LALL_DEV := 12.0, LAL_DEV := 17.0, LAH_DEV := 22.0, LAHH_DEV := 26.0, LAH := 1, LAHH := 1, LALL_TMR.PRE := 90000, LAL_TMR.PRE := 25000, LAH_TMR.PRE := 25000, LAH_TMR.ACC := 25008, LAH_TMR.EN := 1, LAH_TMR.DN := 1, LAHH_TMR.PRE := 90000, LAHH_TMR.ACC := 90007, LAHH_TMR.EN := 1, LAHH_TMR.DN := 1, ForcedValue := 22.0, RawCounts := 18266);   // QUENCH TOWER BASIN LIT
   LC101_AUTO_ONS1 : BOOL := 1;
   LC101_LAHH_MaxTime_TMR : TIMER := (PRE := 180000, ACC := 180006, EN := 1, DN := 1);
   LC101_LAHH_MaxTimeAlm : BOOL := 1;
   LC101_LAHH_MaxTimeMinSP : REAL := 3.0;
   LC101_LT_Raw : REAL := 10.070999;
   LC101_LT_Temp : REAL := 32.10075;
   LC101_MANUAL_ONS1 : BOOL;
   LC101_PD_PV : REAL := 1979.0999;   // SCALER FOR LC 101
   LC101_PD_SCP : SCLP := (Input := 19.790998, InputMax := 100.0, ScaledMax := 10000.0, Output := 1979.0999);
   LC101_PIDE : PID_ENHANCED := (PV := 42.10075, PVEUMax := 100.0, SPProg := 20.0, SPOper := 20.0, SPHLimit := 100.0, RatioProg := 1.0, RatioOper := 1.0, RatioHLimit := 1.0, RatioLLimit := 1.0, CVInitValue := 100.0, CVProg := 99.94373, CVOper := 99.94373, CVEUMax := 30.0, CVEUMin := -30.0, CVHLimit := 100.0, WindupLIn := 1, PGain := 25.0, IGain := 20.0, PVEDerivative := 1, ProgProgReq := 1, ProgManualReq := 1, RTSTime := 1, CVEU := 29.96624, CV := 99.94373, SP := 20.0, SPPercent := 20.0, PVPercent := 42.10075, E := -22.10075, EPercent := -22.10075, InitPrimary := 1, Ratio := 1.0, ProgOper := 1, Manual := 1, DeltaT := 0.01);
   LC101_PIDE_AUTO : BOOL;
   LC101_PIDE_CV_Hold : REAL := 99.94373;
   LC101_SCLP : SCLP := (Input := 100.0, InputMax := 100.0, ScaledMin := 4000.0, ScaledMax := 20000.0, Output := 20000.0);   // QUENCH TRANSFER QUENCH BASIN LEVEL CONTROL OUTPUT SCALER
   LC108_SCLP : SCLP := (Input := 50.0, InputMax := 100.0, ScaledMin := 4000.0, ScaledMax := 20000.0, Output := 12000.0);   // QUENCH BASIN FEED BYPASS LEVEL CONTROL VALVE
   LC205 : LEVEL_CONTROL := (LT := 0.0012497902, LALL_SP := 1.0, LAL_SP := 3.0, LAH_SP := 10.0, LAHH_SP := 14.0, LALL_DEV := 2.0, LAL_DEV := 4.0, LAH_DEV := 9.0, LAHH_DEV := 13.0, LALL := 1, LAL := 1, LALL_TMR.PRE := 5000, LALL_TMR.ACC := 5003, LALL_TMR.EN := 1, LALL_TMR.DN := 1, LAL_TMR.PRE := 5000, LAL_TMR.ACC := 5003, LAL_TMR.EN := 1, LAL_TMR.DN := 1, LAH_TMR.PRE := 5000, LAHH_TMR.PRE := 5000, ForcedValue := 3.0, RawCounts := 4001);   // OVERHEAD CONDENSER BASIN LEVEL CONTROL
   LC205_START_SP : REAL := 9.0;
   LC205_STOP_SP : REAL := 6.0;
   LC205_Totalize_Calc : BOOL;
   LC205_Totalize_End : REAL := 7.95125;
   LC205_Totalize_Gal : REAL;
   LC205_Totalize_Inches : REAL;
   LC205_Totalize_Ini : BOOL;
   LC205_Totalize_Start : REAL;
   LC205_Totalize_Stop : DINT;
   LC205_Totalize_TOF : TIMER := (PRE := 3000, EN := 1, DN := 1);
   LC205_Totalize_Vessel1_Diameter_inches : REAL;
   LC205_Totalize_Vessel1_Gal : REAL;
   LC205_Totalize_Vessel1_Rad_inches : REAL;
   LC205_Totalize_Vessel2_Diameter_inches : REAL;
   LC205_Totalize_Vessel2_Gal : REAL;
   LC205_Totalize_Vessel2_Rad_inches : REAL;
   LC302 : LEVEL_CONTROL := (AUTO_SP := 40.0, LALL_SP := 15.0, LAL_SP := 20.0, LAH_SP := 40.0, LAHH_SP := 45.0, LALL_DEV := 2.0, LAL_DEV := 2.0, LAH_DEV := -1.0, LAHH_DEV := -1.0, LALL := 1, LAL := 1, LALL_TMR.PRE := 5000, LALL_TMR.ACC := 5003, LALL_TMR.EN := 1, LALL_TMR.DN := 1, LAL_TMR.PRE := 5000, LAL_TMR.ACC := 5003, LAL_TMR.EN := 1, LAL_TMR.DN := 1, LAH_TMR.PRE := 5000, LAHH_TMR.PRE := 5000, XA := 1, ForcedValue := 5.0, RawCounts := 3200);   // COALESCER OIL CHAMBER LEVEL CONTROL
   LC302_LT_Raw : REAL := -3.0;
   LC302_SP : SCLP := (Input := 3200.0, InputMin := 4000.0, InputMax := 20000.0, ScaledMax := 60.0, Output := -3.0);   // COALESCER OIL CHAMBER LEVEL TRANSMITTER SCALER
   LC303 : LEVEL_CONTROL := (LALL_SP := 5.0, LAL_SP := 6.0, LAH_SP := 9.0, LAHH_SP := 10.0, LDAH_SP := 5.0, LALL_DEV := 10.0, LAL_DEV := 11.0, LAH_DEV := 4.0, LAHH_DEV := 5.0, LALL := 1, LAL := 1, LALL_TMR.PRE := 5000, LALL_TMR.ACC := 5002, LALL_TMR.EN := 1, LALL_TMR.DN := 1, LAL_TMR.PRE := 5000, LAL_TMR.ACC := 5002, LAL_TMR.EN := 1, LAL_TMR.DN := 1, LAH_TMR.PRE := 5000, LAHH_TMR.PRE := 5000, LDAH_TMR.PRE := 5000);   // COALESCER DIFFEENCE BETWEEN INTERFACE AND AQUEOUS PHASE
   LC303A : LEVEL_CONTROL := (AUTO_SP := 32.0, LT := 19.53058, LALL_SP := 13.0, LAL_SP := 14.0, LAH_SP := 38.0, LAHH_SP := 44.0, LALL_DEV := 1.0, LAL_DEV := 1.0, LAH_DEV := -1.0, LAHH_DEV := -1.0, LALL_TMR.PRE := 60000, LAL_TMR.PRE := 5000, LAH_TMR.PRE := 5000, LAHH_TMR.PRE := 5000, ForcedValue := 40.0);   // AQUEOUS PHASE OF PRIMARY SETTLER
   LC303A_LAHH_PumpShutdownTON : TIMER;
   LC303A_LT_Raw : REAL := 3.53058;
   LC303B : LEVEL_CONTROL := (LT := 19.53058, LALL_SP := 20.0, LAL_SP := 22.0, LAH_SP := 47.0, LAHH_SP := 48.0, LALL_DEV := 21.0, LAL_DEV := 23.0, LAH_DEV := 46.0, LAHH_DEV := 47.0, LALL := 1, LAL := 1, LALL_TMR.PRE := 5000, LALL_TMR.ACC := 5002, LALL_TMR.EN := 1, LALL_TMR.DN := 1, LAL_TMR.PRE := 5000, LAL_TMR.ACC := 5002, LAL_TMR.EN := 1, LAL_TMR.DN := 1, LAH_TMR.PRE := 5000, LAHH_TMR.PRE := 5000, ForcedValue := 45.0);   // INTERFACE LEVEL OF PRIMARY CONDENSER
   LC303B_LT_Raw : REAL := 3.53058;
   LC303C : LEVEL_CONTROL;   // DIFFERENCE BETWEEN INTERFACE AND AQUEOUS PHASE LT 303
   LC304 : LEVEL_CONTROL := (LALL_SP := 5.0, LAL_SP := 10.0, LAH_SP := 25.0, LAHH_SP := 30.0, LALL_DEV := 7.0, LAL_DEV := 8.0, LAH_DEV := 23.0, LAHH_DEV := 28.0, LALL := 1, LAL := 1, LALL_TMR.PRE := 5000, LALL_TMR.ACC := 5003, LALL_TMR.EN := 1, LALL_TMR.DN := 1, LAL_TMR.PRE := 5000, LAL_TMR.ACC := 5003, LAL_TMR.EN := 1, LAL_TMR.DN := 1, LAH_TMR.PRE := 5000, LAHH_TMR.PRE := 5000, ForcedValue := 5.0, RawCounts := 4003);   // SETTLER SECONDARY TANK INTERFACE LEVEL
   LC304_LT_Raw : REAL := 0.009750366;
   LC365_AUTO_SP_START : REAL := 42.0;
   LC365_BLEED_AUTO_SP : REAL := 32.0;
   LC365_BLEED_AUTO_START : BOOL;
   LC365_BLEED_AUTO_START_TON : TIMER := (PRE := 300000);
   LC365_LT : REAL := 19.530605;
   LC370 : LEVEL_CONTROL := (MANUAL := 1, MAN_SP := 50.0, AUTO_SP := 33.0, CO := 50.0, FB := 50.0, PID_CO := 50.0, PV_SETPOINT := 2.0, LT := 19.53058, LALL_SP := 10.0, LAL_SP := 15.0, LAH_SP := 20.0, LAHH_SP := 25.0, LALL_DEV := 11.0, LAL_DEV := 16.0, LAH_DEV := 19.7, LAHH_DEV := 24.7, LALL_TMR.PRE := 5000, LAL_TMR.PRE := 5000, LAH_TMR.PRE := 5000, LAHH_TMR.PRE := 5000);   // WATER MAKE UP FOR PRIMARY SETTLER
   LC370_AUTO_ONS1 : BOOL;
   LC370_AUTO_ONS2 : BOOL := 1;
   LC370_AUTO_SP_START : REAL := 38.0;
   LC370_BLEED_AUTO_SP : REAL := 33.0;
   LC370_Bleed_Makeup_Started : BOOL;
   LC370_FEED_AUTO_START_TON : TIMER;
   LC370_FLOW_TOO_LONG_ALM : BOOL;
   LC370_FLOW_TOO_LONG_RESETPB : BOOL;
   LC370_FLOW_TOO_LONG_TMR : TIMER := (PRE := 600000);
   LC370_HMI_MAKEUP_ENABLE : BOOL;
   LC370_HMI_MAKEUP_REQ : BOOL;
   LC370_HMI_MAKEUP_START_ENABLE : BOOL;
   LC370_HMI_MAKEUP_START_PB : BOOL;
   LC370_HMI_MAKEUP_STOP_PB : BOOL;
   LC370_HMI_VERIFY_PB : BOOL;
   LC370_MAKEUP_AUTO_START_TON : TIMER := (PRE := 60000);
   LC370_MAKUP_AUTO_START_ONS1 : BOOL;
   LC370_MAKUP_AUTO_START_ONS2 : BOOL;
   LC370_MANUAL_ONS1 : BOOL := 1;
   LC370_MAX_TIME_MIN : DINT := 10;
   LC370_Started : BOOL;
   LC370_TOTAl_GAL : REAL := 1113.5907;
   LC370_TOTAl_RESET : BOOL := 1;
   LC370_TOTAl_RESET_PB : BOOL;
   LC370_TOTAl_RESET_TOGGLE : PB_Toggle;
   LC370_TOTALIZE : Totalize := (FlowMeterCV := -0.00031256676, FlowValve := 1, VolAddedLast := 20.853895);
   LC370_TOTALIZE_DISABLE : BOOL;
   LC370_TOTALIZE_EN : BOOL := 1;
   LC370_UNABLE_TO_MAKEUP : BOOL;
   LC_205_SCP : SCLP := (Input := 4001.0, InputMin := 4000.0, InputMax := 20000.0, ScaledMax := 20.0, Output := 0.0012497902);   // OVERHEAD CONDENSER BASIN LEVEL TRANSMITTER SCALER
   LCV101_SCP : SCLP := (Input := 3200.0, InputMin := 4000.0, InputMax := 20000.0, ScaledMax := 100.0, Output := -5.0);
   LCV370_SCLP : SCLP := (Input := 50.0, InputMax := 100.0, ScaledMin := 4000.0, ScaledMax := 20000.0, Output := 12000.0);   // SEPARATOR WATER MAKE UP CONTROL OUTPUT
   LCV370_SCP : SCLP := (Input := 3200.0, InputMin := 4000.0, InputMax := 20000.0, ScaledMax := 100.0, Output := -5.0);
   LCV370_Start : BOOL;
   LevelControlForce : BOOL;
   LevelControlForceONS : BOOL;
   LossOfSignal_mA : DINT := 3810;
   LT101_SCP : SCLP := (Input := 18266.0, InputMin := 4000.0, InputMax := 20000.0, ScaledMax := 36.0, Output := 32.0985);   // QUENCH TOWER BASIN LIT SCALER
   LT303 : REAL := -2.5999994;   // COALESCER OIL CHAMBER LEVEL
   LT303_Probe_Length_Inches : REAL := 52.0;
   LT303_RAW : REAL[5] := ([0] := 5.0863323, [1] := 6.789577, [2] := 6.789577, [4] := 198.37383);   // LT 303 RAW
   LT303_Scale_Param : REAL := 1.9230769;
   LT303_SCP : SCLP := (Input := 3200.0, InputMin := 4000.0, InputMax := 20000.0, ScaledMax := 52.0, Output := -2.5999994);   // COALESCER OIL CHAMBER LEVEL SCALER
   LT304 : REAL := -2.5999994;   // QUENCH COALESCING SEPARATOR SECONDARY CHAMBER LEVEL
   LT304_SCP : SCLP := (Input := 4003.0, InputMin := 4000.0, InputMax := 20000.0, ScaledMax := 52.0, Output := 0.009750366);   // QUENCH COALESCING SEPARATOR SECONDARY CHAMBER LEVEL SCALER
   Major : DINT := 6;
   MATH_TEMP : REAL[30] := ([0] := 15.0);
   MC433A : PUMP_CONTROL := (QI_AUTO := 1, QAS_IAS_TMR.PRE := 10000, LEAD_XFER_TMR.PRE := 5000, RUN_HRS.PRE := 3600000, RUN_HRS.ACC := 3576820, START_DELAY.PRE := 1000);   // HEAT EXCHANGER A
   MC433A_QI_AUTO_OS : BOOL := 1;
   MC433A_QI_MAN_OS : BOOL;
   MC433B : PUMP_CONTROL := (QI_MANUAL := 1, QI_LEAD := 1, START := 1, LEAD_XFER_TMR.PRE := 5000, RUN_HRS.PRE := 3600000, RUN_HRS.ACC := 3576820, START_DELAY.PRE := 1000, START_DELAY.ACC := 1001, START_DELAY.EN := 1, START_DELAY.DN := 1);   // HEAT EXCHANGER 2 STATUS
   MC433B_QI_AUTO_OS : BOOL;
   MC433B_QI_MAN_OS : BOOL := 1;
   MESSAGE_ERROR : DINT;
   Minor : DINT;
   MMI_RESET_PB : BOOL;
   MSG_ConnectionRateSec : DINT := 5;
   MSG_COUNTER : COUNTER := (ACC := 2);
   MSG_ER_AlarmSP : DINT := 1;
   MSG_Group_A : DINT := 1;
   MSG_TimeoutMultiplier : DINT := 1;
   MSG_UnconnectedTimeoutSec : DINT := 5;
   MV115B : ValveControl_TwoWay := (Auto := 1);
   MV301 : ValveControl_TwoWay;
   MV361 : ValveControl_TwoWay := (Status := 1, Auto := 1);
   MV361_AUTO_ONS1 : BOOL := 1;
   MV361_Open : BOOL := 1;
   MV431A : LEVEL_CONTROL;   // QUENCH CONDITIONING HX A INLET VALVE OPEN
   MV431A_OPEN : BOOL;   // H431 HX A INLET VALVE OPEN FAIL OPEN ENERGIZE TO CLOSE
   MV431B : LEVEL_CONTROL;   // QUENCH CONDITIONING HX B INLET VALVE OPEN
   My_Gateway : DINT[4] := ([0] := 192, [1] := 168, [2] := 20, [3] := 1);
        [0]   // Don't touch (auto-filled)
        [1]   // Don't touch (auto-filled)
        [2]   // Don't touch (auto-filled)
        [3]   // !! User to Verify !!
   My_IP_Address : DINT[4] := ([0] := 192, [1] := 168, [2] := 20, [3] := 70);
   My_Subnet : DINT[4] := ([0] := 255, [1] := 255, [2] := 255);
   MyDint : DINT := 8;
   MyTestPID : PID := (CTL := 67146368, SWM := 1, INI := 1, OLH := 1, DVPA := 1, PVHA := 1, SP := 70.0, KP := 1.0, KI := 1.0, MAXS := 4095.0, SO := 100.0, MAXO := 100.0, MINO := 30.0, UPD := 1.0, PV := 53.8125, ERR := 16.1875, OUT := 100.0, MAXI := 4095.0, MAXTIE := 4095.0, DATA[0] := 99.75161, DATA[1] := -21.02564, DATA[2] := 53.8125, DATA[3] := 16.1875, DATA[4] := 70.0, DATA[5] := 0.024420025, DATA[6] := 1.0, DATA[7] := 16.0, DATA[8] := 1.0, DATA[9] := 1.0, DATA[11] := 1.0, DATA[12] := 1.0, DATA[16] := 0.024420025);
   MyTime : DINT[10] := ([0] := 1998, [1] := 1, [2] := 15, [3] := 7, [4] := 15, [5] := 36, [6] := 30479);
   MyToggle : BOOL;
   MyVar : DINT;
   ONE_SHOT : BOOL[32] := ([0] := 1, [4] := 1, [15] := 1, [21] := 1);
        [22]   // LAST USED
   ONE_SHOT_P101B : BOOL := 1;
   ONE_SHOT_P303B : BOOL := 1;
   ONESHOT : DINT;
   option_CartridgeHeaters : BOOL := 1;
   Option_F1_Occupancy : BOOL := 1;   // STATUS FROM UTL PLC 0=DISABLED 1=ENABLED
   P101_NoPumpsAvailAlarm : BOOL := 1;
   P101_NoPumpsAvailTmr : TIMER := (PRE := 5000, ACC := 5007, EN := 1, DN := 1);
   P101_OK_TON : TIMER := (PRE := 10000, ACC := 10003, EN := 1, DN := 1);
   P101_Power : TheTotalizer := (Enable := 1, TotalSecTmr.PRE := 1000, TotalSecTmr.ACC := 179, TotalSecTmr.EN := 1, TotalSecTmr.TT := 1, Minutes := 2.2333333, Totalizer.FlowMeterCV := 1.0079999, Totalizer.FlowValve := 1, Totalizer.VolAddedLast := 1.1345208, Total := 2.311932, Reset := 1, Seconds := 134, Hours := 0.03722222);
   P101A : PUMP_CONTROL := (LOCAL_STATUS := 1, DISABLE := 1, LEAD_DAYS_SP := 15, IAS_SP := 2.0, SIC_MAN_SP := 30.0, SIC_AUTO_SP := 60.0, QAS_IAS_TMR.PRE := 10000, LEAD_XFER_TMR.PRE := 5000, RUN_HRS.PRE := 3600000, START_DELAY.PRE := 5000, ENET_REG_FAULT := 9248, ENET_DATE_TIME[0] := 1998, ENET_DATE_TIME[1] := 1, ENET_DATE_TIME[2] := 15, ENET_DATE_TIME[3] := 7, ENET_DATE_TIME[4] := 15, ENET_DATE_TIME[5] := 33, ENET_DATE_TIME[6] := 770534, Energy := 0.13735998, kWh_Tmr.PRE := 1000, kWh_SampleTime := 1.0, kWh_TimeMultiplier := 3600.0);
   P101A_AmpsFeedback : DINT;
   P101A_BumpStartONS : BOOL;
   P101A_LocalBits : DINT;
   P101A_OK : BOOL;
   P101A_Power : REAL;
   P101A_QI_AUTO_OS : BOOL;
   P101A_QI_MAN_OS : BOOL;
   P101A_SpeedCommand : DINT;
   P101A_SpeedFeedback : DINT;
   P101A_StatusBits : DINT;
   P101B : PUMP_CONTROL := (QI_LEAD := 1, LOCAL_STATUS := 1, DISABLE := 1, LEAD_DAYS_SP := 18, IAS_SP := 2.0, SIC_MAN_SP := 30.0, SIC_AUTO_SP := 60.0, QAS_IAS_TMR.PRE := 10000, LEAD_XFER_TMR.PRE := 5000, RUN_HRS.PRE := 3600000, START_DELAY.PRE := 2000, ENET_REG_FAULT := 9248, ENET_DATE_TIME[0] := 1998, ENET_DATE_TIME[1] := 1, ENET_DATE_TIME[2] := 15, ENET_DATE_TIME[3] := 7, ENET_DATE_TIME[4] := 15, ENET_DATE_TIME[5] := 35, ENET_DATE_TIME[6] := 651918);
   P101B_BumpStartONS : BOOL;
   P101B_OK : BOOL;
   P101B_QI_AUTO_OS : BOOL;
   P101B_QI_MAN_OS : BOOL;
   P101LEADOS : BOOL;
   P205 : PUMP_CONTROL := (QI_LEAD := 1, QI_TRANSFER_LEAD := 1, QI_HOURS := 1, LEAD_DAYS_SP := 365, CUMULATIVE_TM := 1.0, QAS_IAS_TMR.PRE := 10000, LEAD_XFER_TMR.PRE := 5000, RUN_HRS.PRE := 3600000, RUN_HRS.ACC := 2153801);   // OVERHEAD CONDENSER TRANSFER PUMP
   P205_QI_AUTO_OS : BOOL;
   P205_QI_MAN_OS : BOOL;
   P205_START_ONS : BOOL;
   P205_STOP_ONS : BOOL := 1;
   P302_NoPumpsAvailAlarm : BOOL;
   P302_NoPumpsAvailTmr : TIMER;
   P302A : PUMP_CONTROL := (QI_AUTO := 1, LEAD_DAYS_SP := 30, RAMP_SP := 1.0, QAS_IAS_TMR.PRE := 10000, LEAD_XFER_TMR.PRE := 5000, RUN_HRS.PRE := 3600000, SPEED_DELAY.PRE := 1000);
   P302A_OK : BOOL;
   P302A_PumpOut : BOOL;
   P302A_QI_AUTO_ONS1 : BOOL := 1;
   P302A_QI_MAN_ONS1 : BOOL;
   P302B : PUMP_CONTROL := (QI_AUTO := 1, QI_LEAD := 1, YI_LEAD := 1, QI_HOURS := 1, LEAD_DAYS_SP := 30, SIC_AUTO_SP := 40.0, RAMP_SP := 1.0, CUMULATIVE_TM := 1.0, QAS_IAS_TMR.PRE := 10000, LEAD_XFER_TMR.PRE := 5000, RUN_HRS.PRE := 3600000, RUN_HRS.ACC := 374780);
   P302B_OK : BOOL;
   P302B_PumpOut : BOOL;
   P302B_QI_MAN_ONS1 : BOOL;
   P303_NoPumpsAvailAlarm : BOOL;
   P303_NoPumpsAvailTmr : TIMER;
   P303_OK_TON : TIMER := (PRE := 10000, ACC := 10003, EN := 1, DN := 1);
   P303A : PUMP_CONTROL := (LOCAL_STATUS := 1, LEAD_DAYS_SP := 25, IAS_SP := 5.0, SIC_MAN_SP := 30.0, SIC_AUTO_SP := 55.0, RAMP_SP := 5.0, QAS_IAS_TMR.PRE := 20000, LEAD_XFER_TMR.PRE := 5000, RUN_HRS.PRE := 3600000, SPEED_DELAY.PRE := 5000, START_DELAY.PRE := 5000, ENET_REG_FAULT := 9248, ENET_DATE_TIME[0] := 1998, ENET_DATE_TIME[1] := 1, ENET_DATE_TIME[2] := 15, ENET_DATE_TIME[3] := 7, ENET_DATE_TIME[4] := 15, ENET_DATE_TIME[5] := 34, ENET_DATE_TIME[6] := 22353);
   P303A_OK : BOOL;
   P303A_QI_AUTO_OS : BOOL;
   P303A_QI_MAN_OS : BOOL;
   P303A_RPM_SP : INT := 588;
   P303B : PUMP_CONTROL := (QI_LEAD := 1, LOCAL_STATUS := 1, LEAD_DAYS_SP := 22, IAS_SP := 5.0, SIC_MAN_SP := 40.0, SIC_AUTO_SP := 55.0, QAS_IAS_TMR.PRE := 20000, LEAD_XFER_TMR.PRE := 5000, RUN_HRS.PRE := 3600000, START_DELAY.PRE := 2000, ENET_REG_FAULT := 9248, ENET_DATE_TIME[0] := 1998, ENET_DATE_TIME[1] := 1, ENET_DATE_TIME[2] := 15, ENET_DATE_TIME[3] := 7, ENET_DATE_TIME[4] := 15, ENET_DATE_TIME[5] := 36, ENET_DATE_TIME[6] := 54950);
   P303B_OK : BOOL;
   P303B_QI_AUTO_OS : BOOL;
   P303B_QI_MAN_OS : BOOL;
   P305 : PUMP_CONTROL;
   Path_Is_Good : BOOL;
   PC101 : PRESSURE_CONTROL := (PT := 157.34126, PDAH_SP := 11.0, PALL_DEV := 5.0, PAL_DEV := 5.0, PAH_DEV := -5.0, PAHH_DEV := -5.0, PDAH_DEV := 6.0, PAH := 1, PAHH := 1, PDAH := 1, PALL_TMR.PRE := 5000, PAL_TMR.PRE := 5000, PAH_TMR.PRE := 5000, PAH_TMR.ACC := 5003, PAH_TMR.EN := 1, PAH_TMR.DN := 1, PDAH_TMR.PRE := 5000, PDAH_TMR.ACC := 5003, PDAH_TMR.EN := 1, PDAH_TMR.DN := 1, PAHH_TMR.PRE := 5000, PAHH_TMR.ACC := 5003, PAHH_TMR.EN := 1, PAHH_TMR.DN := 1);   // Upper quench tower Diff Pressure
   PC101A : PRESSURE_CONTROL := (PT := 9.368752, PALL_SP := -40.0, PAL_SP := -35.0, PAH_SP := -15.0, PAHH_SP := -5.0, PALL_DEV := -38.0, PAL_DEV := -33.0, PAH_DEV := -17.0, PAHH_DEV := -7.0, PDAH_DEV := -2.0, PAH := 1, PAHH := 1, PALL_TMR.PRE := 300000, PAL_TMR.PRE := 5000, PAH_TMR.PRE := 5000, PAH_TMR.ACC := 5003, PAH_TMR.EN := 1, PAH_TMR.DN := 1, PDAH_TMR.PRE := 5000, PAHH_TMR.PRE := 300000, PAHH_TMR.ACC := 300008, PAHH_TMR.EN := 1, PAHH_TMR.DN := 1, RawCounts := 9045);   // LOWER QUENCH TOWER PRESSURE TRANSMITTER
   PC101B : PRESSURE_CONTROL := (PT := 166.69626, PALL_SP := -40.0, PAL_SP := -35.0, PAH_SP := -15.0, PAHH_SP := -10.0, PALL_DEV := -38.0, PAL_DEV := -33.0, PAH_DEV := -17.0, PAHH_DEV := -12.0, PAH := 1, PAHH := 1, PALL_TMR.PRE := 300000, PAL_TMR.PRE := 5000, PAH_TMR.PRE := 5000, PAH_TMR.ACC := 5003, PAH_TMR.EN := 1, PAH_TMR.DN := 1, PAHH_TMR.PRE := 300000, PAHH_TMR.ACC := 300007, PAHH_TMR.EN := 1, PAHH_TMR.DN := 1, RawCounts := 20487);   // UPPER QUENCH TOWER PRESSURE TRANSMITTER PRESSURE CONTOL
   PC102A : PRESSURE_CONTROL := (PT := 39.044495, PALL_SP := -80.0, PAL_SP := -70.0, PAH_SP := 10.0, PAHH_SP := 15.0, PALL_DEV := -75.0, PAL_DEV := -65.0, PAH_DEV := 5.0, PAHH_DEV := 10.0, PAH := 1, PAHH := 1, PALL_TMR.PRE := 5000, PAL_TMR.PRE := 5000, PAH_TMR.PRE := 5000, PAH_TMR.ACC := 5003, PAH_TMR.EN := 1, PAH_TMR.DN := 1, PAHH_TMR.PRE := 5000, PAHH_TMR.ACC := 5003, PAHH_TMR.EN := 1, PAHH_TMR.DN := 1, RawCounts := 11012);   // QUENCH BASIN TRANSFER PUMP SUCTION PRESSURE CONTROL
   PC102B : PRESSURE_CONTROL := (PT := 1.4099998, PALL_SP := 10.0, PAL_SP := 15.0, PAH_SP := 40.0, PAHH_SP := 45.0, PALL_DEV := 15.0, PAL_DEV := 20.0, PAH_DEV := 35.0, PAHH_DEV := 40.0, PALL := 1, PAL := 1, PALL_TMR.PRE := 5000, PALL_TMR.ACC := 5003, PALL_TMR.EN := 1, PALL_TMR.DN := 1, PAL_TMR.PRE := 5000, PAL_TMR.ACC := 5003, PAL_TMR.EN := 1, PAL_TMR.DN := 1, PAH_TMR.PRE := 5000, PAHH_TMR.PRE := 5000, RawCounts := 4376);   // QUENCH BASIN TRANSFER PUMP DISCHARGE PRESSURE CONTROL
   PC132 : PRESSURE_CONTROL := (AUTO := 1, PT := -10.0, PALL_SP := -50.0, PAL_SP := -40.0, PAH_SP := -20.0, PAHH_SP := -10.0, PALL_DEV := -45.0, PAL_DEV := -35.0, PAH_DEV := -25.0, PAHH_DEV := -15.0, PAH := 1, PALL_TMR.PRE := 5000, PAL_TMR.PRE := 5000, PAH_TMR.PRE := 5000, PAH_TMR.ACC := 5003, PAH_TMR.EN := 1, PAH_TMR.DN := 1, PAHH_TMR.PRE := 5000, XA := 1, RawCounts := 3200, InputMin := 4000, InputMax := 20000);
   PC132_AUTO_Ons : BOOL := 1;
   PC132_AUTO_Ons1 : BOOL;
   PC132_MANUAL_Ons : BOOL;
   PC132_PID : PID := (CTL := -2147450880, EN := 1, INI := 1, MAXS := 4095.0, MAXO := 100.0, MAXI := 4095.0, MAXTIE := 4095.0, DATA[5] := 0.024420025, DATA[6] := 1.0, DATA[16] := 0.024420025);
   PC132_PID_TON : TIMER := (PRE := 500, ACC := 456, EN := 1, TT := 1);
   PC132_SCP : SCLP := (Input := 3200.0, InputMin := 4000.0, InputMax := 20000.0, ScaledMax := 200.0, Output := -10.0);
   PC133 : PRESSURE_CONTROL := (PT := -10.0, PALL_DEV := 5.0, PAL_DEV := 5.0, PAH_DEV := -5.0, PAHH_DEV := -5.0, PALL := 1, PAL := 1, PALL_TMR.PRE := 5000, PALL_TMR.ACC := 5003, PALL_TMR.EN := 1, PALL_TMR.DN := 1, PAL_TMR.PRE := 5000, PAL_TMR.ACC := 5003, PAL_TMR.EN := 1, PAL_TMR.DN := 1, PAH_TMR.PRE := 5000, PAHH_TMR.PRE := 5000, XA := 1, RawCounts := 3200);
   PC133_AUTO_Ons : BOOL;
   PC133_AUTO_Ons1 : BOOL := 1;
   PC133_PID : PID := (CTL := 67141632, SWM := 1, INI := 1, MAXS := 4095.0, MAXO := 100.0, MAXI := 4095.0, MAXTIE := 4095.0, DATA[5] := 0.024420025, DATA[6] := 1.0, DATA[16] := 0.024420025);
   PC133_PID_TON : TIMER := (PRE := 500, ACC := 430, EN := 1, TT := 1);
   PC133_SCP : SCLP := (InputMax := 100.0, ScaledMin := 4000.0, ScaledMax := 20000.0, Output := 4000.0);
   PC134 : PRESSURE_CONTROL := (PT := -10.0, PALL_DEV := 5.0, PAL_DEV := 5.0, PAH_DEV := -5.0, PAHH_DEV := -5.0, PALL := 1, PAL := 1, PALL_TMR.PRE := 5000, PALL_TMR.ACC := 5003, PALL_TMR.EN := 1, PALL_TMR.DN := 1, PAL_TMR.PRE := 5000, PAL_TMR.ACC := 5003, PAL_TMR.EN := 1, PAL_TMR.DN := 1, PAH_TMR.PRE := 5000, PAHH_TMR.PRE := 5000, XA := 1, RawCounts := 3200);
   PC134_AUTO_Ons : BOOL;
   PC134_AUTO_Ons1 : BOOL := 1;
   PC134_PID : PID := (CTL := 67141632, SWM := 1, INI := 1, MAXS := 4095.0, MAXO := 100.0, MAXI := 4095.0, MAXTIE := 4095.0, DATA[5] := 0.024420025, DATA[6] := 1.0, DATA[16] := 0.024420025);
   PC134_PID_TON : TIMER := (PRE := 500, ACC := 420, EN := 1, TT := 1);
   PC134_SCP : SCLP := (InputMax := 100.0, ScaledMin := 4000.0, ScaledMax := 20000.0, Output := 4000.0);
   PC214 : PRESSURE_CONTROL := (AUTO := 1, MAN_SP := 65.0, AUTO_SP := -30.0, CO := 100.0, FB := 100.0, PID_CO := 65.0, PT := 0.30524445, PDAHH_DIFF := 9.063507, PALL_SP := -60.0, PAL_SP := -40.0, PAH_SP := -13.0, PAHH_SP := -10.0, PALL_DEV := -55.0, PAL_DEV := -35.0, PAH_DEV := -18.0, PAHH_DEV := -15.0, PDAH_DEV := 15.0, PDAHH_DEV := 25.0, PAH := 1, PAHH := 1, PALL_TMR.PRE := 5000, PAL_TMR.PRE := 5000, PAH_TMR.PRE := 5000, PAH_TMR.ACC := 5003, PAH_TMR.EN := 1, PAH_TMR.DN := 1, PDAH_TMR.PRE := 10000, PAHH_TMR.PRE := 5000, PAHH_TMR.ACC := 5003, PAHH_TMR.EN := 1, PAHH_TMR.DN := 1, PDAHH_TMR.PRE := 10000, RawCounts := 12332);   // VACUUM SYSTEM PRESSURE TRANSMITTER
   PC214_AUTO_ONS1 : BOOL := 1;
   PC214_MAN_ONS1 : BOOL;
   PC214_PID : PID := (CTL := 33591936, CA := 1, INI := 1, OLH := 1, DVPA := 1, PVHA := 1, SP := -30.0, KP := 20.0, KI := 0.01, BIAS := -33.38745, MAXS := 200.0, MINS := -200.0, SO := 65.0, MAXO := 65.0, MINO := 10.0, UPD := 1.0, PV := 9.368744, ERR := 39.368744, OUT := 65.0, MAXI := 200.0, MINI := -200.0, MAXCV := 100.0, MAXTIE := 4095.0, DATA[0] := 76.22582, DATA[1] := 837.475, DATA[2] := 9.368744, DATA[3] := 39.368744, DATA[4] := -30.0, DATA[5] := 0.25, DATA[6] := 1.0, DATA[7] := 16.0, DATA[8] := 20.0, DATA[9] := 0.01, DATA[11] := 20.0, DATA[12] := 0.01, DATA[15] := 1.0, DATA[16] := 0.024420025);   // QUENCH TOWER EXIT PRESSURE CONTROL VALVE
   PC214_PID_PV : REAL := 9.368752;
   PC214_PID_PV_Select : DINT := 1;   // 0 = PT214 1 = PT101A 2 = PT101B
   PC214_PID_TON : TIMER := (PRE := 100);
   PC214_SCP : SCLP := (Input := 12331.0, InputMin := 4000.0, InputMax := 20000.0, ScaledMin := -45.0, ScaledMax := 42.0, Output := 0.29981232);   // VACUUM SYSTEM PRESSURE TRANSMITTER SCALER
   PC271 : PRESSURE_CONTROL := (AUTO := 1, MAN_SP := 80.0, AUTO_SP := -2.0, CO := 80.0, FB := 80.0, PT := 6.227499, PALL_SP := -20.0, PAL_SP := -15.0, PALL_DEV := -19.0, PAL_DEV := -14.0, PAH_DEV := -1.0, PAHH_DEV := -1.0, PAH := 1, PAHH := 1, PALL_TMR.PRE := 5000, PAL_TMR.PRE := 5000, PAH_TMR.PRE := 5000, PAH_TMR.ACC := 5003, PAH_TMR.EN := 1, PAH_TMR.DN := 1, PAHH_TMR.PRE := 5000, PAHH_TMR.ACC := 5003, PAHH_TMR.EN := 1, PAHH_TMR.DN := 1, RawCounts := 16982);   // VENT HEADER PRESSURE CONTROL
   PC271_AUTO_ONS1 : BOOL := 1;
   PC271_MANUAL_ONS1 : BOOL;
   PC271_PID : PID := (CTL := -2113870592, EN := 1, CA := 1, INI := 1, SPOR := 1, OLL := 1, DVNA := 1, PVLA := 1, SP := -18.0, KP := 100.0, KI := 1.0, MAXS := 10.0, MINS := -10.0, MAXO := 100.0, UPD := 1.0, PV := -14.997725, ERR := -9.997725, MAXI := 20000.0, MINI := 4000.0, MAXTIE := 4095.0, DATA[0] := 24.978563, DATA[1] := -399.81796, DATA[2] := -14.997725, DATA[3] := -9.997725, DATA[4] := -5.0, DATA[5] := 5.0, DATA[6] := 0.00125, DATA[7] := 16.0, DATA[8] := 100.0, DATA[9] := 1.0, DATA[11] := 100.0, DATA[12] := 1.0, DATA[16] := 0.024420025);
   PC271_PID1 : PID := (CTL := 33591936, CA := 1, INI := 1, OLH := 1, DVPA := 1, PVHA := 1, SP := -2.0, KP := 10.0, KI := 0.01, MAXS := 41.0, MINS := -39.99, SO := 80.0, MAXO := 80.0, MINO := 10.0, UPD := 0.2, PV := 6.2317963, ERR := 8.231796, OUT := 80.0, MAXI := 41.0, MINI := -40.0, MAXTIE := 4095.0, DATA[0] := 61.84518, DATA[1] := 913.1358, DATA[2] := 6.2317963, DATA[3] := 8.231796, DATA[4] := -2.0, DATA[5] := 1.2347202, DATA[6] := 0.9998766, DATA[7] := 3.2, DATA[8] := 10.0, DATA[9] := 0.01, DATA[11] := 10.0, DATA[12] := 0.01, DATA[16] := 0.024420025);
   PC271_PID_TON : TIMER := (PRE := 200, ACC := 188, EN := 1, TT := 1);
   PC407A : PRESSURE_CONTROL := (PALL_SP := 10.0, PAL_SP := 20.0, PAH_SP := 70.0, PAHH_SP := 80.0, PDAH_SP := 20.0, PDAHH_SP := 40.0, PALL_DEV := 15.0, PAL_DEV := 25.0, PAH_DEV := 65.0, PAHH_DEV := 75.0, PDAH_DEV := 15.0, PDAHH_DEV := 35.0, PALL := 1, PAL := 1, PALL_TMR.PRE := 5000, PALL_TMR.ACC := 5003, PALL_TMR.EN := 1, PALL_TMR.DN := 1, PAL_TMR.PRE := 5000, PAL_TMR.ACC := 5003, PAL_TMR.EN := 1, PAL_TMR.DN := 1, PAH_TMR.PRE := 5000, PAHH_TMR.PRE := 5000, RawCounts := 4000);   // PRE HX LOW PRESSURE TRANSMITTER
   PC407B : PRESSURE_CONTROL := (PALL_SP := 10.0, PAL_SP := 15.0, PAH_SP := 70.0, PAHH_SP := 80.0, PDAH_SP := 20.0, PDAHH_SP := 40.0, PALL_DEV := 11.0, PAL_DEV := 16.0, PAH_DEV := 69.0, PAHH_DEV := 79.0, PDAH_DEV := 19.0, PDAHH_DEV := 39.0, PALL := 1, PAL := 1, PALL_TMR.PRE := 5000, PALL_TMR.ACC := 5003, PALL_TMR.EN := 1, PALL_TMR.DN := 1, PAL_TMR.PRE := 5000, PAL_TMR.ACC := 5003, PAL_TMR.EN := 1, PAL_TMR.DN := 1, PAH_TMR.PRE := 5000, PAHH_TMR.PRE := 5000, RawCounts := 4000);   // POST HX LOW PRESSURE TRANSMITTER
   PC408 : PRESSURE_CONTROL := (PT := 0.005625725, PALL_DEV := 5.0, PAL_DEV := 5.0, PAH_DEV := -5.0, PAHH_DEV := -5.0, PDAH_DEV := -5.0, PDAHH_DEV := -5.0, PALL := 1, PAL := 1, PAH := 1, PAHH := 1, PALL_TMR.PRE := 5000, PALL_TMR.ACC := 5003, PALL_TMR.EN := 1, PALL_TMR.DN := 1, PAL_TMR.PRE := 5000, PAL_TMR.ACC := 5003, PAL_TMR.EN := 1, PAL_TMR.DN := 1, PAH_TMR.PRE := 5000, PAH_TMR.ACC := 5010, PAH_TMR.EN := 1, PAH_TMR.DN := 1, PDAH_TMR.PRE := 5000, PAHH_TMR.PRE := 5000, PAHH_TMR.ACC := 5010, PAHH_TMR.EN := 1, PAHH_TMR.DN := 1, PDAHH_TMR.PRE := 5000, RawCounts := 4002);
   PC_214_SCP : SCLP := (Input := 9088.0, InputMin := 4000.0, InputMax := 20000.0, ScaledMin := -20.0, ScaledMax := 41.5, Output := -0.4430008);
   PCV214_SCP : SCLP := (Input := 100.0, InputMax := 100.0, ScaledMin := 4000.0, ScaledMax := 20000.0, Output := 20000.0);   // CONDENSER NON CONDENSIBLES CONTROL VALVE OUTPUT SCALER
   PCV271_SCP : SCLP := (Input := 80.0, InputMax := 100.0, ScaledMin := 4000.0, ScaledMax := 20000.0, Output := 16800.0);   // CCONDENSER VENT HEATER CONTROL VALVE OUTPUT
   PDT408_SCP : SCLP := (Input := 4003.0, InputMin := 4000.0, InputMax := 20000.0, ScaledMax := 45.0, Output := 0.00843811);
   PID1_TC215 : PID := (CTL := 33587840, CA := 1, INI := 1, DVPA := 1, PVHA := 1, SP := 40.0, KP := 0.1, KI := 0.1, MAXS := 200.0, SO := 70.172554, MAXO := 100.0, MINO := 30.0, UPD := 0.1, PV := 59.831253, ERR := 19.831253, OUT := 70.172554, MAXI := 200.0, MAXCV := 100.0, MAXTIE := 4095.0, DATA[0] := 69.18099, DATA[1] := 478.65002, DATA[2] := 59.831253, DATA[3] := 19.831253, DATA[4] := 40.0, DATA[5] := 0.5, DATA[6] := 1.0, DATA[7] := 1.6, DATA[8] := 0.1, DATA[9] := 0.1, DATA[11] := 0.1, DATA[12] := 0.1, DATA[15] := 1.0, DATA[16] := 0.024420025);
   PID1_TCV101 : PID := (CTL := 100672768, SWM := 1, CA := 1, OLL := 1, DVNA := 1, PVLA := 1, SP := 20.0, KP := 120.0, KI := 0.1, MAXS := 4095.0, MAXO := 50.0, MINO := 5.0, UPD := 1.0, PV := -1.8000002, ERR := -21.8, OUT := 5.0, MAXI := 4095.0, MAXCV := 100.0, MAXTIE := 4095.0, DATA[0] := 68.899475, DATA[1] := -0.7032968, DATA[2] := -1.8000002, DATA[3] := -21.8, DATA[4] := 20.0, DATA[5] := 0.024420025, DATA[6] := 1.0, DATA[7] := 16.0, DATA[8] := 120.0, DATA[9] := 0.1, DATA[11] := 120.0, DATA[12] := 0.1, DATA[15] := 1.0, DATA[16] := 0.024420025);
   PID_FCV365 : PID := (CTL := 67142272, SWM := 1, INI := 1, DVPA := 1, PVHA := 1, SP := 3.0, KP := 100.0, KI := 200.0, MAXS := 4095.0, MAXO := 60.0, UPD := 0.01, PV := 0.0012500286, ERR := 2.99875, MAXI := 4095.0, MAXCV := 100.0, MAXTIE := 4095.0, DATA[0] := -7.322955, DATA[1] := -0.0004884117, DATA[2] := 0.0012500286, DATA[3] := 2.99875, DATA[4] := 3.0, DATA[5] := 0.024420025, DATA[6] := 1.0, DATA[7] := 0.16, DATA[8] := 100.0, DATA[9] := 200.0, DATA[11] := 100.0, DATA[12] := 200.0, DATA[15] := 1.0, DATA[16] := 0.024420025);
   PID_FCV365_TON : TIMER := (PRE := 10, EN := 1, TT := 1);
   PID_JHE102 : PID := (CTL := 67142784, SWM := 1, INI := 1, DVNA := 1, PVHA := 1, KP := 10.0, KI := 5.0, MAXS := 4095.0, MAXO := 50.0, UPD := 1.0, PV := 61.875, ERR := -61.875, MAXI := 4095.0, MAXTIE := 4095.0, DATA[0] := 15.109891, DATA[1] := -24.175825, DATA[2] := 61.875, DATA[3] := -61.875, DATA[5] := 0.024420025, DATA[6] := 1.0, DATA[7] := 16.0, DATA[8] := 10.0, DATA[9] := 5.0, DATA[11] := 10.0, DATA[12] := 5.0, DATA[16] := 0.024420025);
